				IF (bMinPosMonitoring) THEN
					lrHomingSearchMin := lrMinPos;
				ELSE
					lrHomingSearchMin := -100;
				END_IF
				IF (bMaxPosMonitoring) THEN
					lrHomingSearchMax := lrMaxPos;
				ELSE
					lrHomingSearchMax := 100;
				END_IF
				lrInitTargetSpeed := stAxisParameters.fRefVeloSearch;
				eStep := SP_RunStp1;
			SP_RunStp1 :  (* Move to homing sensor*)
				IF  NOT bHomeSensor THEN
					lrInitTargetPos := lrHomingSearchMin; (*Go in*)
					eStep := SP_RunStp2;
				ELSE
					lrInitTargetPos := lrHomingSearchMax; (*Go out*)
					eStep := SP_RunStp3;
				END_IF
				eInitCommand := AC_MoveAtAbsPos;
			SP_RunStp2 :  (*moving in, search homing*)
				IF afbMoveAbs[iUseBlock].Done THEN
					eCurrentState := AS_InPosition;
				ELSIF afbMoveAbs[iUseBlock].CommandAborted THEN
					iDebugPos := 10;
					eCurrentState := AS_InError;
				ELSIF  bHomeSensor THEN
					lrInitTargetPos := lrHomingSearchMax; (*Go out*)
					eInitCommand := AC_MoveAtAbsPos;
					eStep := SP_RunStp3;
				END_IF
			SP_RunStp3 :(* Moving out, out of sensor*)
				IF afbMoveAbs[iUseBlock].Done THEN
					eCurrentState := AS_InPosition;
				ELSIF afbMoveAbs[iUseBlock].CommandAborted THEN
					iDebugPos := 11;
					eCurrentState := AS_InError;
				ELSIF  NOT bHomeSensor THEN
					lrInitTargetPos := lrHomingSearchMin; (*Go in*)
					eInitCommand := AC_MoveAtAbsPos;
					lrInitTargetSpeed := stAxisParameters.fRefVeloSync;  (* set slow speed*)
					eStep := SP_RunStp4;
				END_IF
			SP_RunStp4 :  (*moving in slowly, search homing*)
				IF afbMoveAbs[iUseBlock].Done THEN
					eCurrentState := AS_InPosition;
				ELSIF afbMoveAbs[iUseBlock].CommandAborted THEN
					iDebugPos := 12;
					eCurrentState := AS_InError;
				ELSIF  bHomeSensor THEN
					lrHomingOffset := ABS(lrCurrentPos);
					lrInitTargetPos := lrCurrentPos; (*Go to home*)
					lrHomingPercent := (lrHomingOffset / lrUnitMotorTurn) * 100;
					eInitCommand := AC_MoveAtAbsPos;
					eStep := SP_RunStp5;
				END_IF
			SP_RunStp5 :(* Wait until position is reached *)
				IF afbMoveAbs[iUseBlock].Done THEN
					eCurrentState := AS_InPosition;
				ELSIF afbMoveAbs[iUseBlock].CommandAborted THEN
					iDebugPos := 13;
					eCurrentState := AS_InError;
				END_IF
			END_CASE
		IF NOT bAxisReady THEN
			iDebugPos := 14;
			eCurrentState := AS_InError;
		END_IF
	AS_MovingLimitNeg:
		CASE eStep OF
			SP_RunStp0 :
				IF bAxisHomed THEN
					eStep := SP_RunStp1;
				ELSE
					eStep := SP_RunStp10;
				END_IF
				lrInitTargetSpeed := stAxisParameters.fRefVeloSearch;
			SP_RunStp1 :  (* Move to Lower limit*)
				IF bMinPosMonitoring THEN
					lrInitTargetPos := lrMinPos;
					eInitCommand := AC_MoveAtAbsPos;
					eStep := SP_RunStp2;
				ELSE
					eCurrentState := AS_InPosition;
					// eCurrentState := AS_InPosition; // TODO : Code Original A enlever com. ?????
				(*ELSIF bNegLimitSwitch THEN // Modif pour test
					eCurrentState := AS_InPosition;
				ELSE
					eCommand := AC_MoveLimitNeg;*)
				END_IF
			SP_RunStp2:
				IF afbMoveAbs[iUseBlock].Done THEN
					eCurrentState := AS_OnLimitNeg;
				ELSIF afbMoveAbs[iUseBlock].CommandAborted THEN
					iDebugPos := 15;
					eCurrentState := AS_InError;
				END_IF
			SP_RunStp10 :  (* Move to LimitNeg sensor*)
				IF  bNegLimitSwitch THEN
					eStep := SP_RunStp13;
				ELSIF lrMoveOutDist = 0 THEN
					eCurrentState := AS_NotHomed;
				ELSE
					lrPosition := lrMoveOutDist+1;
					bSetPosition := TRUE;
					eStep := SP_RunStp11;
				END_IF
				eInitCommand := AC_MoveAtAbsPos;
			SP_RunStp11:
				IF fbSetPosition.Done THEN
					lrInitTargetPos := -lrMoveOutDist;
					eInitCommand := AC_MoveAtRelPos;
					eStep := SP_RunStp12;
				END_IF
			SP_RunStp12:
				IF afbMoveRel[iUseBlock].Done THEN
					eStep := SP_RunStp10;
				ELSIF afbMoveRel[iUseBlock].CommandAborted THEN
					IF  bNegLimitSwitch THEN
						eStep := SP_RunStp13;
					ELSE
						iDebugPos:= 16;
						eCurrentState := AS_InError;
					END_IF
				END_IF
			SP_RunStp13:
				IF bMinPosMonitoring THEN
					lrPosition := lrMinPos+0.5;
					bSetPosition := TRUE;
					eStep := SP_RunStp14;
				ELSE
					eCurrentState := AS_NotHomed;
				END_IF
			SP_RunStp14:
				IF fbSetPosition.Done THEN
					eCurrentState := AS_OnLimitNeg;
				END_IF
			END_CASE
		IF NOT bAxisReady THEN
			iDebugPos := 17;
			eCurrentState := AS_InError;
		END_IF
	AS_OnLimitNeg:
		CASE eCommand OF
			AC_ServoOff:
				eCurrentState := AS_PowerOff;
			AC_Home, AC_Init:
				IF bAxisHomed THEN
					eCurrentState := AS_InPosition;
				ELSE
					eCurrentState := AS_Homing;
				END_IF
		END_CASE
		IF NOT bAxisReady THEN
			iDebugPos := 18;
			eCurrentState := AS_InError;
		END_IF
	AS_Stopping:
		CASE eStep OF
			SP_RunStp0:
				iUseBlock := (iUseBlock + 1) MOD 2;
				bRemoveLimitSecurity := FALSE;
				bHome			:= FALSE;
				bMoveVel 		:= FALSE;
				bMoveAbs 		:= FALSE;
				bMoveRel 		:= FALSE;
				bMoveModulo 	:= FALSE;
				bStop 			:= TRUE;
				bHalt			:= FALSE;
				eStep := SP_RunStp1;
			SP_RunStp1:
				IF afbStop[iUseBlock].Done OR afbStop[iUseBlock].CommandAborted THEN
					iDebugPos := 19;
					eCurrentState := AS_InError;
				END_IF
		END_CASE
	AS_InError:
		CASE eStep OF
			SP_RunStp0:
				ePowerCommand := AC_None;
				bMoveToLimitNegRequest := FALSE;
				bRemoveLimitSecurity := FALSE;
				bServoOn 		:= FALSE;
				bHome			:= TRUE;
				bMoveVel 		:= FALSE;
				bMoveAbs 		:= FALSE;
				bMoveRel 		:= FALSE;
				bMoveModulo 	:= FALSE;
				bStop 			:= FALSE;
				bHalt			:= FALSE;
				bSetPosition 		:= FALSE;
				bAxisHomed		:= FALSE;
				eHomingMode	:= MC_ResetCalibration;
				eStep := SP_RunStp1;
			SP_RunStp1:
				IF fbHome.Done OR fbHome.Error THEN
					bHome := FALSE;
					eStep := SP_RunStp2;
				END_IF
			SP_RunStp2:
				IF bResetErrors THEN
					eCurrentState := AS_Resetting;
				END_IF
		END_CASE
	AS_Resetting:
		IF eCommand = AC_Init OR eCommand = AC_MoveLimitNeg THEN
			ePowerCommand := eCommand;
		END_IF
		CASE eStep OF
			SP_RunStp0:
				IF (eAxisType = AT_AX5000) THEN
					(* For this drive we must use a special drive command for reseting *)
					eStep :=SP_RunStp1;
				ELSE
					eStep :=SP_RunStp10;
				END_IF
			SP_RunStp1:
				fbResetSOE(
					Axis := sAxis,
					Execute := FALSE
				);
				fbResetSOE(
					Axis := sAxis,
					Execute := TRUE
				);
				eStep :=SP_RunStp2;
			SP_RunStp2:
				fbResetSOE(
					Axis := sAxis,
					Execute := FALSE
				);
				IF NOT fbResetSOE.Busy THEN
					IF fbResetSOE.Error THEN
						iDebugPos :=20;
						eCurrentState := AS_InError;
					ELSE
						eStep :=SP_RunStp10;
					END_IF
				END_IF
			SP_RunStp10:
				fbReset(
					Execute 		:= FALSE,
					Axis 		:= sAxis);
				fbReset(
					Execute 		:= TRUE,
					Axis 		:= sAxis);
				eStep :=SP_RunStp11;
			SP_RunStp11:
				fbReset(
					Execute 		:= FALSE,
					Axis 		:= sAxis);
				IF  NOT fbReset.Busy THEN
					IF fbReset.Error THEN
						iDebugPos :=21;
						eCurrentState := AS_InError;
					ELSE
						eCurrentState := AS_PowerOff;
					END_IF
				END_IF
		END_CASE
END_CASE

fbPower(
	Enable			:=	bServoOn,
	Enable_Positive	:=	bServoOn AND NOT bPosLimitSwitch,
	Enable_Negative	:=	bServoOn  AND NOT bNegLimitSwitch,
	Override 			:= 	100.000,
	Axis				:=	sAxis);

fbHome(
	Execute 			:= bHome,
	Position 			:= 0,
	HomingMode		:= eHomingMode,
	bCalibrationCam 	:= bHomeSensor,
	Axis 			:= sAxis);

FOR i:=0 TO 1 DO
	afbMoveAbs[i](
		Execute			:=	bMoveAbs AND iUseBlock = i,
		Position			:=	lrPosition,
		Velocity			:=	lrSpeed,
		Acceleration		:=	lrAcceleration,
		Deceleration		:=	lrDeceleration,
		Jerk 			:=	lrJerk,
		Axis				:=	sAxis);
	afbMoveModulo[i](
		Execute			:=	bMoveModulo AND iUseBlock = i,
		Position			:=	lrPosition,
		Velocity			:=	lrSpeed,
		Acceleration		:=	lrAcceleration,
		Deceleration		:=	lrDeceleration,
		Jerk 			:=	lrJerk,
		Direction    		:=	MC_Shortest_Way,
		Axis				:=	sAxis);
	afbMoveRel[i](
		Execute			:=	bMoveRel AND iUseBlock = i,
		Distance			:=	lrPosition,
		Velocity			:=	lrSpeed,
		Acceleration		:=	lrAcceleration,
		Deceleration		:=	lrDeceleration,
		Jerk 			:=	lrJerk,
		Axis				:=	sAxis);
	afbMoveVel[i](
		Execute			:=	bMoveVel AND iUseBlock = i,
		Velocity			:=	lrSpeed,
		Acceleration		:=	lrAcceleration,
		Deceleration		:=	lrDeceleration,
		Jerk 			:=	lrJerk,
		Direction			:=	eMoveDir,
		Axis				:=	sAxis);
	afbStop[i](
		Execute		:=	bStop AND iUseBlock = i,
		Deceleration	:=	lrDeceleration,
		Jerk 		:=	lrJerk,
		Axis			:=	sAxis);
	afbHalt[i](
		Execute		:=	bHalt AND iUseBlock = i,
		Deceleration	:=	lrDeceleration,
		Jerk 		:=	lrJerk,
		Axis			:=	sAxis);
END_FOR

fbSetPosition(
	Execute		:= bSetPosition,
	Position		:= lrPosition,
	Axis 		:=sAxis);
bSetPosition := FALSE;

fbReadPos(
	Enable 		:= TRUE,
	Axis 		:=sAxis);

fbReadParamTimeToGo(
	Enable 		:= TRUE,
	ReadMode 	:= READMODE_CYCLIC,
	ParameterNumber := AxisRemainingTimeToGo,
	Axis 		:=sAxis
);

(*
fbReadParamModulo(
	Enable 		:= TRUE,
	ReadMode 	:= READMODE_CYCLIC,
	ParameterNumber := AxisEncoderModuloValue,
	Axis 		:=sAxis
);

fbReadParamMinPos(
	Enable 		:= TRUE,
	ReadMode 	:= READMODE_CYCLIC,
	ParameterNumber := SWLimitNeg,
	Axis 		:=sAxis
);

fbReadParamMaxPos(
	Enable 		:= TRUE,
	ReadMode 	:= READMODE_CYCLIC,
	ParameterNumber := SWLimitPos,
	Axis 		:=sAxis
);*)
IF NOT fbReadParameters.Busy THEN
	bReadParameters := NOT bReadParameters;
END_IF

fbReadParameters(
	Execute := 	bReadParameters,
	Parameter := stReadAxisParameters,
	Axis := sAxis
);

fbReadStatus(
	Enable 		:= TRUE,
	Axis 		:=sAxis
);

IF fbReadParamTimeToGo.Valid THEN
	lrRemainingTimeToGo := fbReadParamTimeToGo.Value;
END_IF
(*
IF fbReadParamModulo.Valid THEN
	lrModuloValue := fbReadParamModulo.Value;
END_IF
IF fbReadParamMinPos.Valid THEN
	lrMinPos := fbReadParamMinPos.Value;
END_IF
IF fbReadParamMaxPos.Valid THEN
	lrMaxPos := fbReadParamMaxPos.Value;
END_IF *)
IF fbReadPos.Valid THEN
	lrCurrentPos := fbReadPos.Position;
END_IF

IF fbReadParameters.Done THEN
	stAxisParameters := stReadAxisParameters;
	lrLimitOutSpeed := stAxisParameters.fRefVeloSearch;
	lrModuloValue := stAxisParameters.fEncModuloFactor;
	lrMinPos := stAxisParameters.fEncSoftEndMin;
	lrMaxPos := stAxisParameters.fEncSoftEndMax;
	lrManualSpeed := stAxisParameters.fVeloSlowManual;
	lrFastManualSpeed := stAxisParameters.fVeloFastManual;
	lrRunningSpeed := stAxisParameters.fVeloMaximum ; (* Maximum velocity*)
	bMinPosMonitoring := WORD_TO_BOOL(stAxisParameters.bEncEnableSoftEndMinControl);
	bMaxPosMonitoring := WORD_TO_BOOL(stAxisParameters.bEncEnableSoftEndMaxControl);
	bReadParametersOnce := TRUE;
END_IF

bAxisReady := AxisIsReady(sAxis.NcToPlc.StateDWord);
IF (eAxisType = AT_AX5000) THEN
	sAxis.PlcToNc.ControlDWord := AxisSetAcceptBlockedDriveSignal(sAxis.PlcToNc.ControlDWord, bRemoveLimitSecurity);
	(* sAxis.PlcToNc.ControlDWord.8 := bRemoveLimitSecurity;  Should be remove 01.09.2016 DRE *)
END_IF

(* Error checking*)
IF AxisInErrorState(sAxis.NcToPlc.AxisState) OR fbPower.Error OR fbHome.Error OR fbSetPosition.Error OR fbReadPos.Error OR  (* fbReadParamModulo.Error OR fbReadParamMinPos.Error OR fbReadParamMaxPos.Error OR*) fbReadParameters.Error OR NOT bPowerIsOn THEN
	iDebugPos :=22;
	eCurrentState := AS_InError;
END_IF
FOR i:=0 TO 1 DO
	IF afbMoveAbs[i].Error OR afbMoveModulo[i].Error OR afbMoveRel[i].Error OR afbMoveVel[i].Error OR afbStop[i].Error OR afbHalt[i].Error THEN
		//iDebugPos :=23;
		eCurrentState := AS_InError;
	END_IF
END_FOR

(*Manual Mode Handling *)

stServoButton.Enable := bPowerIsOn AND ((eCurrentState = AS_InPosition) OR (eCurrentState = AS_NotHomed) OR (eCurrentState = AS_PowerOff) OR (eCurrentState = AS_Powering) OR (eCurrentState = AS_OnLimitNeg));
stServoButton.Activate := bServoOn;

iStep := eStep;
iState := eCurrentState;

END_FUNCTION_BLOCK

// ---- POUs/Controls/FB_CheckJack1_2.TcPOU
FUNCTION_BLOCK FB_CheckJack1_2

(*
	Description 	: Bloc fonction de test d'un vérin 1 commande, 2 capteurs
	Auteur		: DLA
	Date		: 26.03.2014
	Version		: 1.00

	Modifications :

*)

VAR_INPUT
	bJackGoOut	: BOOL;
	bJackIsIn	: BOOL;
	bJackIsOut	: BOOL;
	bResetErrors 	: BOOL;
	tTimeOut		: TIME			:= T#400ms;
END_VAR
VAR_OUTPUT
	bJackError	: BOOL;
END_VAR
VAR
	T_Error		: TON;
	RSJackErr	: RS;
	bJackErr		: BOOL;
END_VAR

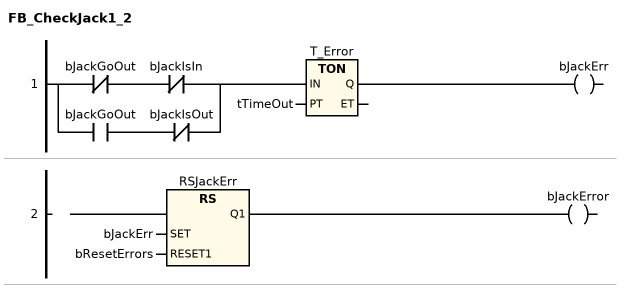
// NETWORK 1
T_Error(IN := NOT bJackGoOut AND NOT bJackIsIn OR bJackGoOut AND NOT bJackIsOut, PT := tTimeOut); // TON
bJackErr := T_Error.Q;

// NETWORK 2
RSJackErr(SET := bJackErr, RESET1 := bResetErrors); // RS
bJackError := RSJackErr.Q1;

END_FUNCTION_BLOCK

// ---- POUs/Controls/FB_VacuumAnalogCheck.TcPOU
FUNCTION_BLOCK FB_VacuumAnalogCheck

(*
	Description 	: Bloc fonction de gestion d'un module de mise sous vide avec niveau de mesure de vide analogique
	Auteur		: DRE
	Date		: 24.08.2016
	Version		: 1.00

	Modifications :

*)

VAR_INPUT
	bEnableVacuum			: BOOL	:= FALSE;			(* Demande d'activation du vacuum *)
	tBlowingTime				: TIME	:= t#200ms;			(* Temps de soufflage à la coupure du vacuum *)
	tVacErrorDelay			: TIME	:= t#400ms;			(* Temps de détection d'une erreur de vide *)
	bReset					: BOOL	:= FALSE;			(* MAZ du bloc en cas d'erreur *)
	iVacuum					: INT;						(* Capteur de vacuum *)
	tWaitVacuumOK			: TIME	:= t#0ms;				(* Temps de détection d'un vide correct *)
	lrVacuumThreshold		: LREAL	:= 9; //-0.7;				(* Seuil de dépression demandée *)
	bDisableVacuumChecking	: BOOL	:= FALSE;
END_VAR
VAR_OUTPUT
	bVacuumOn				: BOOL	:= FALSE;			(* Activation du vacuum *)
	bBlowOn					: BOOL	:= FALSE;			(* Activation du soufflage *)
	bVacuumError			: BOOL	:= FALSE;			(* La demande d'activation s'est terminée par une erreur *)
	lrVacuum				: LREAL	:= 0;					(* Dépression actuelle *)
	bVacuumOK				: BOOL;
	bVacuumCorrect			: BOOL	:= FALSE;			(* La demande d'activation a été bien traitée *)
	bVacuumStable			: BOOL	:= FALSE;			(* Le vacuum est stabilisé *)
END_VAR
VAR
	TInput					: ConverterLinearLimit;
	TVacuum				: FB_Vacuum;
END_VAR
VAR PERSISTENT
	iAnalogMinVoltage		: INT	:= 6500;				(* 1V*)
	iAnalogMaxVoltage 		: INT	:= 31600;				(*5V*)
	lrAnalogMinVacuum		: LREAL	:= 0;					(*kPa or l/min*)
	lrAnalogMaxVacuum 		: LREAL	:= 9.6;					(*kPa or l/min*)
END_VAR

TInput(
	iInput := iVacuum,
	iHardwareMin := iAnalogMinVoltage,
	iHardwareMax := iAnalogMaxVoltage,
	lrSoftwareMin := lrAnalogMinVacuum,
	lrSoftwareMax :=lrAnalogMaxVacuum
	);
lrVacuum := TInput.lrValue;
bVacuumOK := (lrVacuum <= lrVacuumThreshold) AND bEnableVacuum;			// Fonctionnement en vaccum

TVacuum(
	bEnableVacuum := bEnableVacuum,
	tBlowingTime := tBlowingTime,
	tVacErrorDelay := tVacErrorDelay,
	bReset := bReset,
	bVacuumOK := bVacuumOK,
	tWaitVacuumOK := tWaitVacuumOK,
	bDisableVacuumChecking := bDisableVacuumChecking,
	bVacuumOn => bVacuumOn,
	bBlowOn => bBlowOn,
	bVacuumError => bVacuumError,
	bVacuumCorrect => bVacuumCorrect
);

END_FUNCTION_BLOCK

// ---- POUs/utils/ConverterLinearLimit.TcPOU
FUNCTION_BLOCK ConverterLinearLimit
VAR_INPUT
	iInput			: INT;
	iHardwareMin 	: INT;
	iHardwareMax 	: INT;
	lrSoftwareMin 		: LREAL;
	lrSoftwareMax 	: LREAL;
	lrOffset			: LREAL := 0;
END_VAR
VAR_OUTPUT
	lrValue				: LREAL;
	bInputOutOfRange		: BOOL;
END_VAR
VAR
	lrMinOut 			: LREAL;
	lrMaxOut 			: LREAL;
	iHwMinIn 		: LREAL;
	iHwMaxIn		: LREAL;

END_VAR

lrValue := (

			(
				(INT_TO_LREAL(iInput) - INT_TO_LREAL(iHardwareMin))
				/
				(INT_TO_LREAL(iHardwareMax) - INT_TO_LREAL(iHardwareMin))
			)
			*
			( lrSoftwareMax - lrSoftwareMin )
		)
		+ lrSoftwareMin;
IF (lrSoftwareMin > lrSoftwareMax) THEN
	lrMinOut := lrSoftwareMax;
	lrMaxOut := lrSoftwareMin;
ELSE
	lrMinOut := lrSoftwareMin;
	lrMaxOut := lrSoftwareMax;
END_IF
IF lrValue > lrMaxOut THEN lrValue := lrMaxOut; END_IF
IF lrValue < lrMinOut THEN lrValue := lrMinOut; END_IF
lrValue := lrValue + lrOffset;

IF (iHardwareMin > iHardwareMax) THEN
	iHwMinIn := iHardwareMax;
	iHwMaxIn := iHardwareMin;
ELSE
	iHwMinIn := iHardwareMin;
	iHwMaxIn := iHardwareMax;
END_IF
bInputOutOfRange := FALSE;
IF (iInput < iHwMinIn) OR  (iInput > iHwMaxIn) THEN
	bInputOutOfRange:= TRUE;
ELSE
	bInputOutOfRange:= FALSE;
END_IF

END_FUNCTION_BLOCK

// ---- POUs/Controls/FB_Vacuum.TcPOU
FUNCTION_BLOCK FB_Vacuum

(*
	Description 	: Bloc fonction de gestion d'un module de mise sous vide
	Auteur		: DLA
	Date		: 26.03.2014
	Version		: 1.00

	Modifications :

*)

VAR_INPUT
	bEnableVacuum				: BOOL	:= FALSE;			(* Demande d'activation du vacuum *)
	tBlowingTime					: TIME	:= t#200ms;			(* Temps de soufflage à la coupure du vacuum *)
	tVacErrorDelay				: TIME	:= t#400ms;			(* Temps de détection d'une erreur de vide *)
	bReset						: BOOL	:= FALSE;			(* MAZ du bloc en cas d'erreur *)
	bVacuumOK					: BOOL;						(* Capteur de vacuum présent *)
	tWaitVacuumOK				: TIME	:= t#0ms;				(* Temps de détection d'un vide correct *)
	bDisableVacuumChecking		: BOOL	:= FALSE;
END_VAR
VAR_OUTPUT
	bVacuumOn				: BOOL	:= FALSE;			(* Activation du vacuum *)
	bBlowOn					: BOOL	:= FALSE;			(* Activation du soufflage *)
	bVacuumError			: BOOL	:= FALSE;			(* La demande d'activation s'est terminée par une erreur *)
	bVacuumCorrect			: BOOL	:= FALSE;			(* La demande d'activation a été bien traitée *)
	bVacuumStable			: BOOL	:= FALSE;			(* Le vacuum est stabilisé *)
END_VAR
VAR
	bVacuumIsOK			: BOOL	:= FALSE;			(* Information que le vacuum est OK *)
	TVacError				: TON;
	TVacOK					: TON;
	TBlow					: TON;
	TVacCut					: TON;
END_VAR

(*La commande de vacuum est directement reliée à la requête*)
bVacuumOn := bEnableVacuum;

bVacuumIsOK := bVacuumOK;

(*On fait tourner les timers de détection de vacuum et de soufflage*)
TBlow(IN:=NOT bEnableVacuum,PT:=tBlowingTime);
TVacOK(IN:=bEnableVacuum AND bVacuumOK,PT:=tWaitVacuumOK);
TVacCut(IN := NOT bEnableVacuum AND NOT bVacuumOK AND NOT bBlowOn, PT := t#100ms);
bVacuumStable := TVacOK.Q;

IF bEnableVacuum THEN
	bBlowOn := FALSE;
	(*On détecte si le vacuum ne s'établit pas assez vite*)
	TVacError(IN:=NOT (bVacuumOK OR bDisableVacuumChecking) ,PT:=tVacErrorDelay);
	IF bDisableVacuumChecking THEN
		bVacuumCorrect := TRUE;
	ELSE
		bVacuumCorrect := TVacOK.Q;
	END_IF
	IF  TVacError.Q AND NOT bVacuumOK THEN
		bVacuumError := TRUE;
	END_IF
ELSE
	(*On contrôle que le vacuum s'est bien coupé aprés le soufflage*)
	bBlowOn := NOT TBlow.Q;
	bVacuumCorrect := NOT bVacuumOK AND NOT bBlowOn;
	bVacuumCorrect := TVacCut.Q;
	TVacError(IN:=bVacuumOK AND NOT bBlowOn,PT:=tVacErrorDelay);
	IF TVacError.Q THEN
		bVacuumError := TRUE;
	END_IF
END_IF
IF bVacuumCorrect THEN
	TVacError(IN:=FALSE);
END_IF
IF bReset AND bVacuumError THEN
	TBlow(IN:= FALSE);
	TVacError(IN:=FALSE);
	bVacuumOn := FALSE;
	bBlowOn := FALSE;
	bReset := FALSE;
	bVacuumError := FALSE;
END_IF

END_FUNCTION_BLOCK

// ---- POUs/utils/ComputeVisionPos.TcPOU
FUNCTION_BLOCK ComputeVisionPos
VAR_INPUT
	THead			: TPositionXY;
	lrAngle			: LREAL;
END_VAR
VAR_OUTPUT
	TOffsetPos				: TPositionXYTheta;
END_VAR
VAR
	lrHypotenuse		: LREAL;
	lrAngle1			: LREAL;
	lrAngle2			: LREAL;
	lrAngleVision		: LREAL;
END_VAR

lrAngleVision := LMOD((lrAngle* -1) + 180 + 45,180);
lrHypotenuse := SQRT(EXPT(THead.lrX,2) + EXPT(THead.lrY,2));
IF THead.lrX = 0 THEN
	lrAngle1 := 90;
ELSE
	lrAngle1 := RAD_TO_DEG(ATAN(ABS(THead.lrY) / ABS(THead.lrX)));
END_IF
IF THead.lrX < 0 AND THead.lrY >= 0 THEN
	lrAngle1 := lrAngle1 + 90;
ELSIF THead.lrX < 0 AND THead.lrY < 0 THEN
	lrAngle1 := lrAngle1 + 180;
ELSIF THead.lrX >= 0 AND THead.lrY < 0 THEN
	lrAngle1 := lrAngle1 + 270;
END_IF
lrAngle2 := lrAngleVision - lrAngle1;
TOffsetPos.lrX := COS(DEG_TO_RAD(lrAngle2)) * -lrHypotenuse;
TOffsetPos.lrY := SIN(DEG_TO_RAD(lrAngle2)) * lrHypotenuse;
TOffsetPos.lrTheta := lrAngleVision;

END_FUNCTION_BLOCK

// ---- POUs/utils/InitNewPartData.TcPOU
FUNCTION InitNewPartData : TPartData
VAR_INPUT
END_VAR
VAR
	TPartData	: TPartData;
	i			: INT;
	j			: INT;
END_VAR

TPartData.bPartPresent := FALSE;
TPartData.bToReject := FALSE;
TPartData.bSample := FALSE;
FOR i := 0 TO 1 DO
	FOR j := 0 TO 1 DO
		TPartData.abHasPearls[i,j] := FALSE;
		TPartData.abBadPearling[i,j] := FALSE;
		TPartData.abPearlingDone[i,j] := FALSE;
		TPartData.anLastPearlIndexDone[i,j] := 0;
	END_FOR
END_FOR
TPartData.dwPlateInQRCode := 0;
TPartData.iPlateInPos := 0;
TPartData.dwPlateOutQRCode := 0;
TPartData.iPlateOutPos := 0;
TPartData.ePartSide := PS_SUS;
TPartData.dwProductionTime := 0;
TPartData.dwProductionInTime := 0;
TPartData.dwProductionOutTime := 0;
InitNewPartData := TPartData;

END_FUNCTION

// ---- POUs/utils/GetLoaderTeachedAxisFromAxis.TcPOU
FUNCTION GetLoaderTeachedAxisFromAxis : TLoaderTeachedAxis
VAR_INPUT
	eAxis	: TLoaderAxis;
END_VAR
VAR
END_VAR

CASE eAxis OF
	LA_X:
		GetLoaderTeachedAxisFromAxis := LTA_X;
	LA_Y:
		GetLoaderTeachedAxisFromAxis := LTA_Y;
	LA_Z1:
		GetLoaderTeachedAxisFromAxis := LTA_Z;
	LA_Z2:
		GetLoaderTeachedAxisFromAxis := LTA_Z;
	LA_THETA:
		GetLoaderTeachedAxisFromAxis := LTA_THETA;
END_CASE

END_FUNCTION

// ---- POUs/Handlers/TableHdl.TcPOU
FUNCTION_BLOCK TableHdl

(*
	Description 	: Function bloc to handle rotation table
	Author		: DLA
	Date		: 18.08.2014
	Version		: 1.00

	Modifications :

*)

VAR_INPUT
	bEnable						: BOOL;
	bPowerOn					: BOOL;
	bHomeTable					: BOOL;
	bHomeBrush					: BOOL;
	bLimitPosBrush				: BOOL;
	bLimitNegBrush				: BOOL;
	bResetErrors				: BOOL;
	iTableVacuumPos1Flow		: INT;
	iTableVacuumPos2Flow		: INT;
	iTableVacuumPos3Flow		: INT;
	iTableVacuumPos4Flow		: INT;
	bTableLocked				: BOOL;
	bTableNotLocked				: BOOL;
	bAspirationIsUp				: BOOL;
	bAspirationIsDown			: BOOL;
	bCheckVacuum4Rotation		: BOOL;
	eCommand					: TModuleCommands;
	bStopReq					: BOOL;
	bPauseReq					: BOOL;
	sInGiveToLoader				: TTaker;
	sInTakeFromLoader			: TGiver;
	eRunCommand				: TRunCmdTable;
	bLayeringWithTwoParts		: BOOL;
	bManInterlock				: BOOL;
	sVaccumSettings				: TVaccumSettings;
	iPartialGiveTakeTime			: INT;
	bVisionConfig					: BOOL;
	bCleanBrushIsUp				: BOOL;
	bCleanBrushIsDown				: BOOL;
END_VAR
VAR_OUTPUT
	bModuleError					: BOOL;
	bAspirationError				: BOOL;
	bIndexTableError				: BOOL;
	bPlate1VacuumError			: BOOL;
	bPlate2VacuumError			: BOOL;
	bPlate3VacuumError			: BOOL;
	bPlate4VacuumError			: BOOL;
	bTableAxisError				: BOOL;
	bBrushAxisError				: BOOL;
	bAspirationGoDown			: BOOL;
	bAspirationGoUp				: BOOL;
	bIndexTable					: BOOL;
	bAspirationBrushOn			: BOOL;
	bActivatePlate1Vacuum		: BOOL;
	bActivatePlate1Blowing		: BOOL;
	bActivatePlate2Vacuum		: BOOL;
	bActivatePlate2Blowing		: BOOL;
	bActivatePlate3Vacuum		: BOOL;
	bActivatePlate3Blowing		: BOOL;
	bActivatePlate4Vacuum		: BOOL;
	bActivatePlate4Blowing		: BOOL;
	bVacuumErrForRotation		: BOOL;
	bVacuumNotOk4Pearling		: BOOL;
	eSideOnLoader				: TTableSide;
	sOutGiveToLoader			: TGiver;
	sOutTakeFromLoader			: TTaker;
	eRunStatus					: TRunStatus;
	bManInterlockOut			: BOOL;
	aiPearlsVacuumFlow			: ARRAY[0..1] OF INT;
	bMoveCleanBrushDown			: BOOL;
	bCleanBrushError			: BOOL;
END_VAR
VAR_IN_OUT
	sCurrentState					: TModuleData;
	sRunData					: TRunDataTable;
	TManualCmd					: TManTable;
	sTableAxisRef				: AXIS_REF;
	sBrushAxisRef				: AXIS_REF;
END_VAR
VAR CONSTANT
	lrSafeTolerance 					:LREAL := 1;											(* Tolerance for safety axis *)
	lrPositionTolerance 				: LREAL := 0.1;
END_VAR
VAR PERSISTENT
	alrWorkingPos				: ARRAY [0..1] OF LREAL := [0,180];		(* Working position of table CW / CCW *)
	alrBrushParkPos				: ARRAY [0..1] OF LREAL := [0,0];
	alrBrushWorkPos				: ARRAY [0..1] OF LREAL := [90,90];
	alrBrushSpeed				: ARRAY [0..1] OF LREAL := [80,100]; 	// initial value [40,60];
	lrTableJogStep				: LREAL					:= 5;
	iNbOfCleaning				: INT					:= 1;
	lrBrushJogStep				: LREAL					:= 5;
	alrVacuumThreshold			: ARRAY[0..3] OF LREAL	:= [8,8,8,8];// [-0.65,-0.65,-0.65,-0.65];
	lrTableCleanSpeed			: LREAL					:= 30;
END_VAR
VAR
	i							: INT;
	abEnablePlateVacuum			: ARRAY[0..3] OF BOOL;
	abPlateVacuumOK			: ARRAY[0..3] OF BOOL;
	abPlateVacuumError			: ARRAY[0..3] OF BOOL;
	abForceBlowing				: ARRAY[0..3] OF BOOL;
	abDisableVacuumChecking	: ARRAY[0..3] OF BOOL;
	abActivatePlateBlowing		: ARRAY[0..3] OF BOOL;
	abActivatePlateVacuum		: ARRAY[0..3] OF BOOL;
	aiTableVacuumPosFlow	: ARRAY[0..3] OF INT;
	eMoveTableAxisCommand		: TAxisCommands	:= AC_None;
	eMoveBrushAxisCommand		: TAxisCommands	:= AC_None;
	lrTableTargetPos				: LREAL;
	lrBrushTargetPos				: LREAL;
	lrCurrentTableMoveSpeed		: LREAL;
	lrRunTableMoveSpeed		: LREAL;
	lrCurrentBrushMoveSpeed		: LREAL;
	TAspiration					: FB_CheckJack2_2;
	TIndexTable					: FB_CheckJack1_2;
	TCleanBrush				: FB_CheckJack1_2;
	aTPlateVacuum				: ARRAY[0..3] OF  FB_VacuumAnalogCheck;
	TAxisTable					: StdAxis;
	TAxisBrush					: StdAxis;
	iGiveTakePos				: INT;
	iCleaningPos					: INT;
	iCleaningCycle				: INT;
	iOffsetPosNotTakeGive		: INT;
	iTargetWorkingPos			: INT;
	TGiveTakeTimer				: TON;
	bPartialGiveTake				: BOOL;
	bTableOkToMove			: BOOL;
	TVacuumTimer				: TON;
	eLastStatus 					: TModuleStatus := MS_Stopped;
	tPartialGiveTakeTime			: TIME;
	bCleanAfterTurn				: BOOL;
	eCleaningStep				: TModuleSteps;
	bDoCleaningSeq				: BOOL;
	bDoCleaningOnMoveSeq		: BOOL;
	bStopCleaningOnMoveSeq		: BOOL;
	iStep						: INT;
END_VAR

IF (NOT sCurrentState.bStepMode) THEN
	sCurrentState.bWaitStep := FALSE;
END_IF

(* Optimize code *)
aiTableVacuumPosFlow[0] := iTableVacuumPos1Flow;
aiTableVacuumPosFlow[1] := iTableVacuumPos2Flow;
aiTableVacuumPosFlow[2] := iTableVacuumPos3Flow;
aiTableVacuumPosFlow[3] := iTableVacuumPos4Flow;
tPartialGiveTakeTime := INT_TO_TIME(iPartialGiveTakeTime);

IF eLastStatus<>sCurrentState.eStatus THEN
	IF eLastStatus=MS_Manual THEN
		(*Leave manual mode, redefine part present base on vacuum *)
		IF NOT abEnablePlateVacuum[0] THEN
			sRunData.aTPartData[0,0,TS_A].bPartPresent := FALSE;
			sRunData.aTPartData[0,1,TS_A].bPartPresent := FALSE;
		END_IF
		IF NOT abEnablePlateVacuum[1] THEN
			sRunData.aTPartData[1,0,TS_A].bPartPresent := FALSE;
			sRunData.aTPartData[1,1,TS_A].bPartPresent := FALSE;
		END_IF
		IF NOT abEnablePlateVacuum[2] THEN
			sRunData.aTPartData[0,0,TS_B].bPartPresent := FALSE;
			sRunData.aTPartData[0,1,TS_B].bPartPresent := FALSE;
		END_IF
		IF NOT abEnablePlateVacuum[3] THEN
			sRunData.aTPartData[1,0,TS_B].bPartPresent := FALSE;
			sRunData.aTPartData[1,1,TS_B].bPartPresent := FALSE;
		END_IF
	END_IF
	IF eLastStatus=MS_Running OR sCurrentState.eStatus=MS_Manual THEN
		(* Set vaccum base on part present, Vacuum can be disable if take part has failed*)
		IF NOT bVisionConfig THEN
			abEnablePlateVacuum[0] := sRunData.aTPartData[0,0,TS_A].bPartPresent OR sRunData.aTPartData[0,1,TS_A].bPartPresent;
		END_IF
		abEnablePlateVacuum[1] := sRunData.aTPartData[1,0,TS_A].bPartPresent OR sRunData.aTPartData[1,1,TS_A].bPartPresent;
		abEnablePlateVacuum[2] := sRunData.aTPartData[0,0,TS_B].bPartPresent OR sRunData.aTPartData[0,1,TS_B].bPartPresent;
		abEnablePlateVacuum[3] := sRunData.aTPartData[1,0,TS_B].bPartPresent OR sRunData.aTPartData[1,1,TS_B].bPartPresent;
	END_IF
	eLastStatus := sCurrentState.eStatus;
END_IF
IF NOT bLayeringWithTwoParts THEN
	sRunData.aTPartData[0,1,TS_A].bPartPresent := FALSE;
	sRunData.aTPartData[1,1,TS_A].bPartPresent := FALSE;
	sRunData.aTPartData[0,1,TS_B].bPartPresent := FALSE;
	sRunData.aTPartData[1,1,TS_B].bPartPresent := FALSE;
END_IF

CASE eCommand OF
	MC_NoCmd :
		CASE sCurrentState.eStatus OF
			MS_Init :
				CASE sCurrentState.eStep OF
					SP_InitStp1 :
						(* Init all synchros *)
						FOR i := 0 TO 3 DO
							abForceBlowing[i] := FALSE;
							abDisableVacuumChecking[i] := FALSE;
							(*abEnablePlateVacuum[i] := TRUE;*)
						END_FOR
						bMoveCleanBrushDown := FALSE;
						bAspirationBrushOn := FALSE;
						TVacuumTimer(IN := FALSE);
						sCurrentState.eStep := SP_InitStp2;
					SP_InitStp2 :
						TVacuumTimer(IN := TRUE, PT := t#0s);
						IF TVacuumTimer.Q THEN
							IF NOT bVisionConfig THEN
								abEnablePlateVacuum[0] := sRunData.aTPartData[0,0,TS_A].bPartPresent OR sRunData.aTPartData[0,1,TS_A].bPartPresent;
							END_IF
							abEnablePlateVacuum[1] := sRunData.aTPartData[1,0,TS_A].bPartPresent OR sRunData.aTPartData[1,1,TS_A].bPartPresent;
							abEnablePlateVacuum[2] := sRunData.aTPartData[0,0,TS_B].bPartPresent OR sRunData.aTPartData[0,1,TS_B].bPartPresent;
							abEnablePlateVacuum[3] := sRunData.aTPartData[1,0,TS_B].bPartPresent OR sRunData.aTPartData[1,1,TS_B].bPartPresent;
							IF bLayeringWithTwoParts THEN
							 	abDisableVacuumChecking[0] := sRunData.aTPartData[0,0,TS_A].bPartPresent XOR sRunData.aTPartData[0,1,TS_A].bPartPresent;
								abDisableVacuumChecking[1] := sRunData.aTPartData[1,0,TS_A].bPartPresent XOR sRunData.aTPartData[1,1,TS_A].bPartPresent;
								abDisableVacuumChecking[2] := sRunData.aTPartData[0,0,TS_B].bPartPresent XOR sRunData.aTPartData[0,1,TS_B].bPartPresent;
								abDisableVacuumChecking[3] := sRunData.aTPartData[1,0,TS_B].bPartPresent XOR sRunData.aTPartData[1,1,TS_B].bPartPresent;
							END_IF
							IF sCurrentState.bInitDone THEN
								sCurrentState.eStep := SP_InitStp50;
							ELSE
								sCurrentState.eStep := SP_InitStp3;
							END_IF
						END_IF
					SP_InitStp3 :
						(* Put the clean brush in the waiting position - Raise the aspiration - Lower index table *)
						bAspirationGoDown := FALSE;
						bIndexTable := FALSE;
						sCurrentState.eStep := SP_InitStp4;
					SP_InitStp4 :
						(* Wait until all jacks are in position *)
						IF  bAspirationIsUp AND bTableNotLocked THEN
							sCurrentState.eStep := SP_InitStp5;
						END_IF
					SP_InitStp5 :
						eMoveBrushAxisCommand := AC_Init;
						eMoveTableAxisCommand := AC_Init;
						sCurrentState.eStep := SP_InitStp6;
					SP_InitStp6 :
						IF TAxisTable.eCurrentState =  AS_InPosition AND TAxisBrush.eCurrentState =  AS_InPosition THEN
							lrTableTargetPos := alrWorkingPos[0];
							lrRunTableMoveSpeed := TAxisTable.lrRunningSpeed;
							eMoveTableAxisCommand := AC_MoveAtAbsPos;
							lrBrushTargetPos := alrBrushParkPos[0];
							(* During init always use low speed *)
							lrCurrentBrushMoveSpeed := alrBrushSpeed[0];
							eMoveBrushAxisCommand := AC_MoveAtAbsPos;
							sCurrentState.eStep := SP_InitStp7;
						END_IF
					SP_InitStp7 :
						(* Wait until init position is reached *)
						IF TAxisTable.eCurrentState =  AS_InPosition AND TAxisBrush.eCurrentState =  AS_InPosition THEN
							(* Index table *)
							bIndexTable := TRUE;
							sCurrentState.eStep := SP_InitStp8;
						END_IF
					SP_InitStp8 :
						IF bTableLocked THEN
							bAspirationGoDown := TRUE;
							sCurrentState.eStep := SP_InitStp9;
						END_IF
					SP_InitStp9 :
						IF  bAspirationIsDown THEN
							eSideOnLoader := TS_A;
							sCurrentState.eStep := SP_InitStp99;
						END_IF
					SP_InitStp50 :
						lrBrushTargetPos := alrBrushParkPos[0];
						eMoveBrushAxisCommand := AC_MoveAtAbsPos;
						sCurrentState.eStep := SP_InitStp51;
					SP_InitStp51 :
						IF TAxisBrush.eCurrentState =  AS_InPosition THEN
							sCurrentState.eStep := SP_InitStp99;
						END_IF
					SP_InitStp99 : (* Leave init *)
						sCurrentState.eStep := SP_RunStp1;
						sCurrentState.eStatus := MS_Ready;
						bDoCleaningSeq:= FALSE;
						bDoCleaningOnMoveSeq:= FALSE;
						bStopCleaningOnMoveSeq:= FALSE;
						eCleaningStep := SP_RunStp1;
						sCurrentState.bInitDone := TRUE;
				END_CASE
			MS_Running :
				IF (NOT sCurrentState.bWaitStep) THEN
					(* Cleaning sequence *)
					CASE eCleaningStep OF
						SP_RunStp1 :
							IF bUse103171OptimB5CleanOn1Move THEN
								eCleaningStep := SP_RunStp50;
							ELSE
								eCleaningStep := SP_RunStp10;
							END_IF
						SP_RunStp10 :
							IF bDoCleaningSeq THEN
								IF eSideOnLoader = TS_B THEN
									iCleaningPos := 2;
								ELSE
									iCleaningPos := 0;
								END_IF
								FOR i := 0 TO 1 DO
									IF NOT sRunData.aTPartData[i, 0, eSideOnLoader].bPartPresent AND NOT sRunData.aTPartData[i, 1, eSideOnLoader].bPartPresent THEN
										abForceBlowing[i + iCleaningPos] := TRUE;
									END_IF
								END_FOR
								bAspirationBrushOn := TRUE;
								bMoveCleanBrushDown := TRUE;
								iCleaningCycle := 0;
								eCleaningStep := SP_RunStp12;
							END_IF
						SP_RunStp11:
							IF iCleaningCycle < iNbOfCleaning THEN
								lrBrushTargetPos := alrBrushWorkPos[0];
								eMoveBrushAxisCommand := AC_MoveAtAbsPos;
								eCleaningStep := SP_RunStp12;
							ELSE
								eCleaningStep := SP_RunStp14;
							END_IF
						SP_RunStp12:
							IF (TAxisBrush.eCurrentState = AS_InPosition) THEN
								lrBrushTargetPos := alrBrushWorkPos[1];
								eMoveBrushAxisCommand := AC_MoveAtAbsPos;
								eCleaningStep := SP_RunStp13;
							END_IF
						SP_RunStp13:
							IF (TAxisBrush.eCurrentState = AS_InPosition) THEN
								iCleaningCycle := iCleaningCycle + 1;
								eCleaningStep := SP_RunStp11;
							END_IF
						SP_RunStp14:
							IF (TAxisBrush.eCurrentState = AS_InPosition) THEN
								lrBrushTargetPos := alrBrushParkPos[0];
								eMoveBrushAxisCommand := AC_MoveAtAbsPos;
								eCleaningStep := SP_RunStp15;
							END_IF
						SP_RunStp15:
							IF (TAxisBrush.eCurrentState = AS_InPosition) THEN
								eCleaningStep := SP_RunStp16;
							END_IF
						SP_RunStp16:
							FOR i := iCleaningPos TO iCleaningPos+1 DO
								abForceBlowing[i] := FALSE;
							END_FOR
							bAspirationBrushOn := FALSE;
							bMoveCleanBrushDown := FALSE;
							bDoCleaningSeq:= FALSE;
							eCleaningStep := SP_RunStp10;
						SP_RunStp50:							
							IF bDoCleaningSeq THEN
								eCleaningStep := SP_RunStp60;
							ELSIF bDoCleaningOnMoveSeq THEN
								eCleaningStep := SP_RunStp80;
							END_IF
						SP_RunStp60 :
							IF eSideOnLoader = TS_B THEN
								iCleaningPos := 1;
							ELSE
								iCleaningPos := 0;
							END_IF
							FOR i := 0 TO 1 DO
								IF NOT sRunData.aTPartData[i, 0, eSideOnLoader].bPartPresent AND NOT sRunData.aTPartData[i, 1, eSideOnLoader].bPartPresent THEN
									abForceBlowing[i + iCleaningPos] := TRUE;
								END_IF
							END_FOR
							bAspirationBrushOn := TRUE;
							bMoveCleanBrushDown := TRUE;
							eCleaningStep := SP_RunStp61;
						SP_RunStp61: 
							(* Go to other position *)
							IF TAxisBrush.lrCurrentPos < (alrBrushParkPos[0] + 1) THEN
								lrBrushTargetPos := alrBrushWorkPos[1];
							ELSE
								lrBrushTargetPos := alrBrushWorkPos[0];
							END_IF
							lrCurrentBrushMoveSpeed := alrBrushSpeed[1];
							eMoveBrushAxisCommand := AC_MoveAtAbsPos;
							eCleaningStep := SP_RunStp62;
						SP_RunStp62:
							IF (TAxisBrush.eCurrentState = AS_InPosition) THEN
								(* Move to final position *)
								lrBrushTargetPos := alrBrushWorkPos[iCleaningPos];
								eMoveBrushAxisCommand := AC_MoveAtAbsPos;
								eCleaningStep := SP_RunStp63;
							END_IF
						SP_RunStp63:
							IF (TAxisBrush.eCurrentState = AS_InPosition) THEN
								bAspirationBrushOn := FALSE;
								bMoveCleanBrushDown := FALSE;
								bDoCleaningSeq:= FALSE;
								eCleaningStep := SP_RunStp50;
							END_IF
						SP_RunStp80:
							bAspirationBrushOn := TRUE;
							bDoCleaningOnMoveSeq := FALSE;
							IF eSideOnLoader = TS_B THEN
								iCleaningPos := 0;
							ELSE
								iCleaningPos := 1;
							END_IF
							eCleaningStep := SP_RunStp81;
						SP_RunStp81:
							IF bStopCleaningOnMoveSeq THEN
								bAspirationBrushOn := FALSE;
								bStopCleaningOnMoveSeq := FALSE;
								eCleaningStep := SP_RunStp50;
							END_IF
					END_CASE
					CASE sCurrentState.eStep OF
						SP_RunStp1:
							eRunStatus := RS_WaitRequest;
							CASE eRunCommand OF
								RCT_None:
									IF bStopReq  THEN
										sCurrentState.eStatus := MS_Ready;
									ELSIF bPauseReq THEN
										sCurrentState.eStatus := MS_Paused;
									END_IF
								RCT_TakePart:
									sOutTakeFromLoader.bHasTaken := FALSE;
									sOutTakeFromLoader.bHasNotTaken := FALSE;
									sOutTakeFromLoader.bReadyToTake := TRUE;
									sCurrentState.eStep := SP_RunStp10;
								RCT_GivePart:
									sOutGiveToLoader.bHasGiven := FALSE;
									sOutGiveToLoader.bPartDataReady := FALSE;
									sCurrentState.eStep := SP_RunStp20;
								RCT_Turn:
									bCleanAfterTurn := FALSE;
									sCurrentState.eStep := SP_RunStp30;
								RCT_Clean:
									sCurrentState.eStep := SP_RunStp40;
								RCT_TurnAndClean:
									bCleanAfterTurn := TRUE;
									sCurrentState.eStep := SP_RunStp30;
							END_CASE
							IF sCurrentState.eStep<> SP_RunStp1 THEN eRunStatus := RS_ProcessRequest1; END_IF
						SP_RunStp10 :  (*Take Part*)
							IF sInTakeFromLoader.bPartDataReady THEN
								sRunData.aTPartData[ sRunData.iGiveTakeLayeringPosition, sRunData.iGiveTakeLayeringOffsetPosition, eSideOnLoader] := sInTakeFromLoader.TPartData;
								sRunData.aTPartData[sRunData.iGiveTakeLayeringPosition, sRunData.iGiveTakeLayeringOffsetPosition, eSideOnLoader].bPartPresent := FALSE;
								sCurrentState.eStep := SP_RunStp11;
							END_IF
						SP_RunStp11 :
							IF eSideOnLoader = TS_B THEN
								iGiveTakePos := sRunData.iGiveTakeLayeringPosition + 2;
							ELSE
								iGiveTakePos := sRunData.iGiveTakeLayeringPosition;
							END_IF
							iOffsetPosNotTakeGive := ((sRunData.iGiveTakeLayeringOffsetPosition + 1) MOD 2);
							abEnablePlateVacuum[iGiveTakePos] := TRUE;
							sOutTakeFromLoader.bReadyToTake := TRUE;
							IF bLayeringWithTwoParts AND NOT sRunData.aTPartData[sRunData.iGiveTakeLayeringPosition, iOffsetPosNotTakeGive, eSideOnLoader].bPartPresent THEN
								bPartialGiveTake:= TRUE;
							ELSE
								bPartialGiveTake:= FALSE;
							END_IF
							abDisableVacuumChecking[iGiveTakePos] := TRUE;
							sCurrentState.eStep := SP_RunStp12;
						SP_RunStp12 :
							(* Wait until loader has given *)
							IF sInTakeFromLoader.bHasGiven THEN
								sRunData.aTPartData[sRunData.iGiveTakeLayeringPosition, sRunData.iGiveTakeLayeringOffsetPosition, eSideOnLoader].bPartPresent := TRUE;
								abDisableVacuumChecking[iGiveTakePos] := TRUE;
								TGiveTakeTimer(IN:= FALSE);
								sCurrentState.eStep := SP_RunStp13;
							END_IF
						SP_RunStp13 :
							(* Check if the part is on Layering *)
							TGiveTakeTimer(IN:=TRUE, PT := tPartialGiveTakeTime );
							IF NOT bPartialGiveTake THEN
								IF bRejectPartWithVacuumErrorOnTable THEN
									TVacuumTimer(IN := FALSE);
									sCurrentState.eStep := SP_RunStp16;
								ELSE
									sOutTakeFromLoader.bHasTaken := TRUE;
									sCurrentState.eStep := SP_RunStp14;
								END_IF
							ELSIF TGiveTakeTimer.Q THEN
								sOutTakeFromLoader.bHasTaken := TRUE;
								sCurrentState.eStep := SP_RunStp1;
							END_IF
						SP_RunStp14 :
							IF NOT sInTakeFromLoader.bHasGiven THEN
								abDisableVacuumChecking[iGiveTakePos] := FALSE;
								sCurrentState.eStep := SP_RunStp15;
							END_IF
						SP_RunStp15 :
							IF aTPlateVacuum[iGiveTakePos].bVacuumCorrect THEN
								sCurrentState.eStep := SP_RunStp1;
							END_IF
						SP_RunStp16 :
							(* Wait until vacuum correct or vacuum error *)
							TVacuumTimer(IN := TRUE, PT := aTPlateVacuum[iGiveTakePos].tVacErrorDelay);
							IF aTPlateVacuum[iGiveTakePos].bVacuumStable THEN
								sOutTakeFromLoader.bHasTaken := TRUE;
								sCurrentState.eStep := SP_RunStp14;
							ELSIF TVacuumTimer.Q THEN
								sOutTakeFromLoader.bHasNotTaken := TRUE;
								abEnablePlateVacuum[iGiveTakePos] := FALSE;
								abDisableVacuumChecking[iGiveTakePos] := FALSE;
								sCurrentState.eStep := SP_RunStp17;
							END_IF
						SP_RunStp17 :
							IF NOT sInTakeFromLoader.bHasGiven THEN
								sRunData.aTPartData[sRunData.iGiveTakeLayeringPosition, sRunData.iGiveTakeLayeringOffsetPosition, eSideOnLoader].bPartPresent := FALSE;
								sCurrentState.eStep := SP_RunStp1;
							END_IF
						SP_RunStp20 : (*Give Part*)
							sOutGiveToLoader.TPartData := sRunData.aTPartData[sRunData.iGiveTakeLayeringPosition, sRunData.iGiveTakeLayeringOffsetPosition, eSideOnLoader];
							sOutGiveToLoader.bPartDataReady := TRUE;
							sCurrentState.eStep := SP_RunStp21;
						SP_RunStp21 :
							IF sInGiveToLoader.bReadyToTake THEN
								IF eSideOnLoader = TS_B THEN
									iGiveTakePos := sRunData.iGiveTakeLayeringPosition + 2;
								ELSE
									iGiveTakePos := sRunData.iGiveTakeLayeringPosition;
								END_IF
								abEnablePlateVacuum[iGiveTakePos] := FALSE;
								sCurrentState.eStep := SP_RunStp22;
							END_IF
						SP_RunStp22 :
							(* Check if laying vacuum is disabled *)
							IF aTPlateVacuum[iGiveTakePos].bVacuumCorrect THEN
								sOutGiveToLoader.bHasGiven := TRUE;
								sCurrentState.eStep := SP_RunStp23;
							END_IF
						SP_RunStp23 :
							(* Check if right loader has taken the plate *)
							IF sInGiveToLoader.bHasTaken THEN
								sRunData.aTPartData[sRunData.iGiveTakeLayeringPosition, sRunData.iGiveTakeLayeringOffsetPosition, eSideOnLoader].bPartPresent := FALSE;
								sCurrentState.eStep := SP_RunStp1;
							END_IF
						SP_RunStp30:
							bTableOkToMove := TRUE;
							FOR i:=0 TO 3 DO
								IF NOT aTPlateVacuum[iGiveTakePos].bVacuumCorrect THEN
									bTableOkToMove := FALSE;
								END_IF
							END_FOR
							IF bTableOkToMove THEN
								bAspirationGoDown := FALSE;
								IF bCleanAfterTurn AND bUse103171OptimB5CleanOnBothSide THEN
									bDoCleaningOnMoveSeq := TRUE;
									eCleaningStep := SP_RunStp1;
								END_IF
								sCurrentState.eStep := SP_RunStp31;
							END_IF
						SP_RunStp31 :
							IF  bAspirationIsUp THEN
								bIndexTable := FALSE;
								sCurrentState.eStep := SP_RunStp32;
							END_IF
						SP_RunStp32 :
							IF  bTableNotLocked AND NOT bDoCleaningOnMoveSeq THEN
								IF eSideOnLoader = TS_A THEN
									iTargetWorkingPos := 1;
								ELSE
									iTargetWorkingPos := 0;
								END_IF
								lrTableTargetPos := alrWorkingPos[iTargetWorkingPos];
								IF bCleanAfterTurn AND bUse103171OptimB5CleanOnBothSide THEN
									lrRunTableMoveSpeed := lrTableCleanSpeed;
								ELSE
									lrRunTableMoveSpeed := TAxisTable.lrRunningSpeed;
								END_IF
								eSideOnLoader := TS_Moving;
								eMoveTableAxisCommand := AC_MoveAtAbsPos;
								sCurrentState.eStep := SP_RunStp35;
							END_IF
						SP_RunStp35 :
							IF NOT bDoCleaningSeq THEN
								(* Wait until position is reached *)
								IF (TAxisTable.eCurrentState = AS_InPosition) THEN
									(* Index table *)
									bIndexTable := TRUE;
									(* And clean if needed *)
									IF bUse103171OptimB5CleanOnBothSide THEN
										bStopCleaningOnMoveSeq := TRUE;
									ELSIF bCleanAfterTurn THEN
										bDoCleaningSeq := TRUE;
										eCleaningStep := SP_RunStp1;
									END_IF
									sCurrentState.eStep := SP_RunStp36;
								END_IF
							END_IF
						SP_RunStp36 :
							IF bTableLocked THEN
								bAspirationGoDown := TRUE;
								sCurrentState.eStep := SP_RunStp37;
							END_IF
						SP_RunStp37 :
							IF  bAspirationIsDown THEN
								eRunStatus := RS_ProcessRequest2;
								IF NOT bDoCleaningSeq THEN
									IF iTargetWorkingPos = 0 THEN
										eSideOnLoader := TS_A;
									ELSE
										eSideOnLoader := TS_B;
									END_IF
									sCurrentState.eStep := SP_RunStp1;
								END_IF
							END_IF
						SP_RunStp40:
							IF NOT bDoCleaningSeq THEN
								bDoCleaningSeq := TRUE;
								eCleaningStep := SP_RunStp1;
								sCurrentState.eStep := SP_RunStp41;
							END_IF
						SP_RunStp41:
							IF NOT bDoCleaningSeq THEN
								sCurrentState.eStep := SP_RunStp1;
							END_IF
					END_CASE
				END_IF
			MS_Manual :
				TManualCmd.TAxisTable.Home.Enable := NOT bManInterlock AND bAspirationIsUp AND bTableNotLocked AND ((TAxisTable.eCurrentState = AS_InPosition) OR (TAxisTable.eCurrentState = AS_NotHomed));
				TManualCmd.TAxisTable.MoveBw.Enable := NOT bManInterlock AND bAspirationIsUp AND bTableNotLocked AND (TAxisTable.eCurrentState = AS_InPosition)  AND (TAxisTable.lrCurrentPos-lrTableJogStep >= TAxisTable.lrMinPos);
				TManualCmd.TAxisTable.MoveFw.Enable := NOT bManInterlock AND bAspirationIsUp AND bTableNotLocked AND (TAxisTable.eCurrentState = AS_InPosition) AND (TAxisTable.lrCurrentPos+lrTableJogStep <= TAxisTable.lrMaxPos);
				TManualCmd.TAxisTableLoading12Pos.MoveToTeach.Enable := NOT bManInterlock AND bAspirationIsUp AND bTableNotLocked AND (TAxisTable.eCurrentState = AS_InPosition) AND alrWorkingPos[0] >= TAxisTable.lrMinPos AND alrWorkingPos[0] <= TAxisTable.lrMaxPos;
				TManualCmd.TAxisTableLoading34Pos.MoveToTeach.Enable := NOT bManInterlock AND bAspirationIsUp AND bTableNotLocked AND (TAxisTable.eCurrentState = AS_InPosition) AND alrWorkingPos[1] >= TAxisTable.lrMinPos AND alrWorkingPos[1] <= TAxisTable.lrMaxPos;
				TManualCmd.TAxisTable.CurrentPos := TAxisTable.lrCurrentPos;

				TManualCmd.TAxisBrush.Home.Enable := NOT bManInterlock AND bTableLocked AND ((TAxisBrush.eCurrentState = AS_InPosition) OR (TAxisBrush.eCurrentState = AS_NotHomed));
				TManualCmd.TAxisBrush.MoveBw.Enable := NOT bManInterlock AND bTableLocked AND (TAxisBrush.eCurrentState = AS_InPosition)  AND (TAxisBrush.lrCurrentPos-lrBrushJogStep >= TAxisBrush.lrMinPos) ;
				TManualCmd.TAxisBrush.MoveFw.Enable := NOT bManInterlock AND bTableLocked AND (TAxisBrush.eCurrentState = AS_InPosition)  AND (TAxisBrush.lrCurrentPos+lrBrushJogStep <= TAxisBrush.lrMaxPos) ;
				FOR i:= 0 TO 1 DO
					TManualCmd.aTAxisBrushParkPos[i].MoveToTeach.Enable := NOT bManInterlock AND bTableLocked AND (TAxisBrush.eCurrentState = AS_InPosition)  AND alrBrushParkPos[i] >= TAxisBrush.lrMinPos AND alrBrushParkPos[i] <= TAxisBrush.lrMaxPos;
					TManualCmd.aTAxisBrushWorkPos[i].MoveToTeach.Enable := NOT bManInterlock AND bTableLocked AND (TAxisBrush.eCurrentState = AS_InPosition)  AND alrBrushWorkPos[i] >= TAxisBrush.lrMinPos AND alrBrushWorkPos[i] <= TAxisBrush.lrMaxPos;;
				END_FOR
				TManualCmd.TAxisBrush.CurrentPos := TAxisBrush.lrCurrentPos;

				TManualCmd.TAspirationDown.Enable := NOT bManInterlock AND  (((TAxisTable.eCurrentState = AS_InPosition) AND (ABS(TAxisTable.lrCurrentPos - alrWorkingPos[0])<lrPositionTolerance) OR  (ABS(TAxisTable.lrCurrentPos - alrWorkingPos[1])<lrPositionTolerance)) OR bAspirationGoDown);
				TManualCmd.TIndexTable.Enable := ((TAxisTable.eCurrentState = AS_InPosition) AND (ABS(TAxisTable.lrCurrentPos - alrWorkingPos[0])<lrPositionTolerance) OR  (ABS(TAxisTable.lrCurrentPos - alrWorkingPos[1])<lrPositionTolerance)) OR bIndexTable;

				IF bTableLocked AND eSideOnLoader = TS_Moving THEN
					IF (ABS(TAxisTable.lrCurrentPos - alrWorkingPos[0])<lrPositionTolerance) THEN
						eSideOnLoader := TS_A;
					ELSIF (ABS(TAxisTable.lrCurrentPos - alrWorkingPos[1])<lrPositionTolerance) THEN
						eSideOnLoader := TS_B;
					END_IF
				ELSIF NOT bTableLocked THEN
					eSideOnLoader := TS_Moving;
				END_IF
				FOR i:= 0 TO 3 DO
					TManualCmd.alrVaccumValue[i] := aTPlateVacuum[i].lrVacuum;
				END_FOR
				TManualCmd.TPlate1Vacuum.Enable := TAxisTable.eCurrentState <> AS_Moving AND TAxisTable.eCurrentState <> AS_Stopping AND TAxisTable.eCurrentState <> AS_Homing  AND
													TAxisBrush.eCurrentState <> AS_Moving AND TAxisBrush.eCurrentState <> AS_Stopping AND TAxisBrush.eCurrentState <> AS_Homing;
				TManualCmd.TPlate2Vacuum.Enable := TManualCmd.TPlate1Vacuum.Enable;
				TManualCmd.TPlate3Vacuum.Enable := TManualCmd.TPlate1Vacuum.Enable;
				TManualCmd.TPlate4Vacuum.Enable :=TManualCmd.TPlate1Vacuum.Enable;

				TManualCmd.TAspirationBrush.Enable := TRUE;
				TManualCmd.TCleanBrushDown.Enable := TRUE;
				bManInterlockOut := NOT (eSideOnLoader <> TS_Moving AND
								 ((TAxisBrush.lrCurrentPos <= (alrBrushParkPos[0]+lrSafeTolerance)) OR (TAxisBrush.lrCurrentPos >= (alrBrushParkPos[1]-lrSafeTolerance))) AND
								TAxisBrush.bAxisHomed AND bAspirationIsDown);


				CASE sCurrentState.eStep OF
					SP_ManualStp0 :
						// Table
						TManualCmd.TAxisTable.Home.Activate := FALSE;
						TManualCmd.TAxisTable.JogStep := lrTableJogStep;
						TManualCmd.TAxisTable.MoveBw.Activate := FALSE;
						TManualCmd.TAxisTable.MoveFw.Activate := FALSE;
						TManualCmd.TAxisTableLoading12Pos.MoveToTeach.Activate := FALSE;
						TManualCmd.TAxisTableLoading12Pos.Teach := FALSE;
						TManualCmd.TAxisTableLoading34Pos.MoveToTeach.Activate := FALSE;
						TManualCmd.TAxisTableLoading34Pos.Teach := FALSE;
						// Brush
						TManualCmd.TAxisBrush.Home.Activate := FALSE;
						TManualCmd.TAxisBrush.JogStep := lrBrushJogStep;
						TManualCmd.TAxisBrush.MoveBw.Activate := FALSE;
						TManualCmd.TAxisBrush.MoveFw.Activate := FALSE;
						FOR i:= 0 TO 1 DO
							TManualCmd.aTAxisBrushParkPos[i].MoveToTeach.Activate := FALSE;
							TManualCmd.aTAxisBrushParkPos[i].Teach := FALSE;
							TManualCmd.aTAxisBrushWorkPos[i].MoveToTeach.Activate := FALSE;
							TManualCmd.aTAxisBrushWorkPos[i].Teach := FALSE;
						END_FOR
						FOR i:= 0 TO 3 DO
							TManualCmd.alrVaccumThershold[i] := alrVacuumThreshold[i];
						END_FOR


						TManualCmd.TPlate1Vacuum.Activate := abEnablePlateVacuum[0];
						TManualCmd.TPlate2Vacuum.Activate := abEnablePlateVacuum[1];
						TManualCmd.TPlate3Vacuum.Activate := abEnablePlateVacuum[2];
						TManualCmd.TPlate4Vacuum.Activate := abEnablePlateVacuum[3];
						TManualCmd.TAspirationDown.Activate := bAspirationGoDown;
						TManualCmd.TIndexTable.Activate := bIndexTable;

						TManualCmd.TAspirationBrush.Activate := bAspirationBrushOn;
						TManualCmd.TCleanBrushDown.Activate := bMoveCleanBrushDown;
						sCurrentState.eStep := SP_ManualStp1;
					SP_ManualStp1 :
						IF bStopReq THEN
							sCurrentState.eStatus := MS_Stopped;
						ELSE
							FOR i:= 0 TO 1 DO
								TManualCmd.aTAxisBrushWorkPos[i].TeachedPos := alrBrushWorkPos[i];
								TManualCmd.aTAxisBrushParkPos[i].TeachedPos := alrBrushParkPos[i];
							END_FOR
							TManualCmd.TAxisTableLoading12Pos.TeachedPos := alrWorkingPos[0];
							TManualCmd.TAxisTableLoading34Pos.TeachedPos := alrWorkingPos[1];
							IF (lrTableJogStep <> TManualCmd.TAxisTable.JogStep) THEN
								lrTableJogStep := TManualCmd.TAxisTable.JogStep;
							END_IF
							IF TManualCmd.TAxisTableLoading12Pos.Teach THEN
								alrWorkingPos[0] := TAxisTable.lrCurrentPos;
								TManualCmd.TAxisTableLoading12Pos.Teach := FALSE;
							END_IF
							IF TManualCmd.TAxisTableLoading34Pos.Teach THEN
								alrWorkingPos[1] := TAxisTable.lrCurrentPos;
								TManualCmd.TAxisTableLoading34Pos.Teach := FALSE;
							END_IF
							IF TManualCmd.TAxisTableLoading12Pos.MoveToTeach.Activate THEN
								lrTableTargetPos := alrWorkingPos[0];
								sCurrentState.eStep := SP_ManualStp10;
							ELSIF TManualCmd.TAxisTableLoading34Pos.MoveToTeach.Activate THEN
								lrTableTargetPos := alrWorkingPos[1];
								sCurrentState.eStep := SP_ManualStp10;
							ELSIF TManualCmd.TAxisTable.MoveBw.Activate THEN
								lrTableTargetPos := TAxisTable.lrCurrentPos - lrTableJogStep;
								sCurrentState.eStep := SP_ManualStp10;
							ELSIF TManualCmd.TAxisTable.MoveFw.Activate THEN
								lrTableTargetPos := TAxisTable.lrCurrentPos + lrTableJogStep;
								sCurrentState.eStep := SP_ManualStp10;
							END_IF
							IF TManualCmd.TAxisTable.Home.Activate AND sCurrentState.eStep = SP_ManualStp1 THEN
								sCurrentState.eStep := SP_ManualStp20;
							END_IF


							IF (lrBrushJogStep <> TManualCmd.TAxisBrush.JogStep) THEN
								lrBrushJogStep := TManualCmd.TAxisBrush.JogStep;
							END_IF
							FOR i:= 0 TO 1 DO
								IF TManualCmd.aTAxisBrushParkPos[i].Teach THEN
									alrBrushParkPos[i] := TAxisBrush.lrCurrentPos;
									TManualCmd.aTAxisBrushParkPos[i].Teach := FALSE;
								END_IF
								IF TManualCmd.aTAxisBrushWorkPos[i].Teach THEN
									alrBrushWorkPos[i] := TAxisBrush.lrCurrentPos;
									TManualCmd.aTAxisBrushWorkPos[i].Teach := FALSE;
								END_IF
								IF TManualCmd.aTAxisBrushParkPos[i].MoveToTeach.Activate THEN
									lrBrushTargetPos := alrBrushParkPos[i];
									sCurrentState.eStep := SP_ManualStp15;
								ELSIF TManualCmd.aTAxisBrushWorkPos[i].MoveToTeach.Activate THEN
									lrBrushTargetPos := alrBrushWorkPos[i];
									sCurrentState.eStep := SP_ManualStp15;
								END_IF
							END_FOR
							IF TManualCmd.TAxisBrush.MoveBw.Activate THEN
								lrBrushTargetPos := TAxisBrush.lrCurrentPos - lrBrushJogStep;
								sCurrentState.eStep := SP_ManualStp15;
							ELSIF TManualCmd.TAxisBrush.MoveFw.Activate THEN
								lrBrushTargetPos := TAxisBrush.lrCurrentPos + lrBrushJogStep;
								sCurrentState.eStep := SP_ManualStp15;
							END_IF

							IF TManualCmd.TAxisBrush.Home.Activate AND sCurrentState.eStep = SP_ManualStp1 THEN
								sCurrentState.eStep := SP_ManualStp25;
							END_IF
							FOR i:= 0 TO 3 DO
								IF TManualCmd.alrVaccumThershold[i] <> alrVacuumThreshold[i] THEN
									alrVacuumThreshold[i] := TManualCmd.alrVaccumThershold[i];
								END_IF
							END_FOR

							bAspirationGoDown := TManualCmd.TAspirationDown.Activate;
							bIndexTable := TManualCmd.TIndexTable.Activate;
							abEnablePlateVacuum[0] := TManualCmd.TPlate1Vacuum.Activate;
							abEnablePlateVacuum[1] := TManualCmd.TPlate2Vacuum.Activate;
							abEnablePlateVacuum[2] := TManualCmd.TPlate3Vacuum.Activate;
							abEnablePlateVacuum[3] := TManualCmd.TPlate4Vacuum.Activate;
						END_IF
					SP_ManualStp10 : (*Move Table *)
						eMoveTableAxisCommand := AC_MoveAtAbsPos;
						sCurrentState.eStep := SP_ManualStp11;
					SP_ManualStp11:
						CASE TAxisTable.eCurrentState OF
							AS_InPosition, AS_InError:
								TManualCmd.TAxisTableLoading12Pos.MoveToTeach.Activate := FALSE;
								TManualCmd.TAxisTableLoading34Pos.MoveToTeach.Activate := FALSE;
								TManualCmd.TAxisTable.MoveFw.Activate := FALSE;
								TManualCmd.TAxisTable.MoveBw.Activate := FALSE;
								sCurrentState.eStep := SP_ManualStp1;
						END_CASE
					SP_ManualStp15: (*Move Brush *)
						eMoveBrushAxisCommand := AC_MoveAtAbsPos;
						sCurrentState.eStep := SP_ManualStp16;
					SP_ManualStp16:
						CASE TAxisBrush.eCurrentState OF
							AS_InPosition, AS_InError:
								FOR i := 0 TO 1 DO
									TManualCmd.aTAxisBrushParkPos[i].MoveToTeach.Activate := FALSE;
									TManualCmd.aTAxisBrushWorkPos[i].MoveToTeach.Activate := FALSE;
								END_FOR
								TManualCmd.TAxisBrush.MoveFw.Activate := FALSE;
								TManualCmd.TAxisBrush.MoveBw.Activate := FALSE;
								sCurrentState.eStep := SP_ManualStp1;
						END_CASE
					SP_ManualStp20 :  (* Init Table *)
						eMoveTableAxisCommand := AC_Home;
						sCurrentState.eStep := SP_ManualStp21;
					SP_ManualStp21 :
						CASE TAxisTable.eCurrentState OF
							AS_InPosition:
								lrTableTargetPos := alrWorkingPos[0];
								eMoveTableAxisCommand := AC_MoveAtAbsPos;
								sCurrentState.eStep := SP_ManualStp22;
							AS_InError:
								sCurrentState.eStep := SP_ManualStp1;
								TManualCmd.TAxisTable.Home.Activate := FALSE;
						END_CASE
					SP_ManualStp22 :
						CASE TAxisTable.eCurrentState OF
							AS_InPosition, AS_InError:
								sCurrentState.eStep := SP_ManualStp1;
								TManualCmd.TAxisTable.Home.Activate := FALSE;
						END_CASE
					SP_ManualStp25 :  (* Init Brush*)
						eMoveBrushAxisCommand := AC_Home;
						sCurrentState.eStep := SP_ManualStp26;
					SP_ManualStp26 :
						CASE TAxisBrush.eCurrentState OF
							AS_InPosition:
								lrBrushTargetPos := alrBrushParkPos[0];
								eMoveBrushAxisCommand := AC_MoveAtAbsPos;
								sCurrentState.eStep := SP_ManualStp27;
							AS_InError:
								sCurrentState.eStep := SP_ManualStp1;
								TManualCmd.TAxisBrush.Home.Activate := FALSE;
						END_CASE
					SP_ManualStp27 :(* Wait until init position is reached *)
						CASE TAxisBrush.eCurrentState OF
							AS_InPosition, AS_InError:
								sCurrentState.eStep := SP_ManualStp1;
								TManualCmd.TAxisBrush.Home.Activate := FALSE;
						END_CASE
				END_CASE
				bAspirationBrushOn := TManualCmd.TAspirationBrush.Activate;
				bMoveCleanBrushDown := TManualCmd.TCleanBrushDown.Activate;
			MS_Paused:
				IF bStopReq THEN
					sCurrentState.eStatus := MS_Ready;
				END_IF
		END_CASE
	MC_Init :
		sCurrentState.eStep := SP_InitStp1;
		sCurrentState.eStatus := MS_Init;
	MC_Run :
		sCurrentState.eStatus := MS_Running;
	MC_Manual :
		sCurrentState.bInitDone := FALSE;
		sCurrentState.eStatus := MS_Manual;
		sCurrentState.eStep := SP_ManualStp0;
	MC_Stop :
		sCurrentState.eStatus := MS_Stopped;
END_CASE


IF (NOT bPowerOn) THEN
	bAspirationGoDown := TRUE;
	bIndexTable := FALSE;
	TManualCmd.TAspirationDown.Activate := bAspirationGoDown;
	TManualCmd.TIndexTable.Activate := bIndexTable;
END_IF

IF bResetErrors THEN
	bVacuumErrForRotation := FALSE;
	sCurrentState.bInError := FALSE;
END_IF

IF (sCurrentState.eStatus <> MS_Manual) THEN
	IF (eMoveTableAxisCommand <> AC_None ) AND
		NOT bAspirationIsUp OR NOT bTableNotLocked THEN
		bTableAxisError := TRUE;
		eMoveTableAxisCommand := AC_None;
	END_IF
END_IF

(* Table Axis *)
IF (sCurrentState.eStatus = MS_Manual) THEN
	lrCurrentTableMoveSpeed := TAxisTable.lrManualSpeed;
ELSE
	lrCurrentTableMoveSpeed := lrRunTableMoveSpeed;
END_IF
TAxisTable(
	eCommand		:= eMoveTableAxisCommand,
	lrTargetPos		:= lrTableTargetPos,
	lrTargetSpeed	:= lrCurrentTableMoveSpeed,
	sAxis			:= sTableAxisRef,
	bResetErrors		:= bResetErrors,
	bHomeSensor	:= bHomeTable,
	bPowerIsOn		:= bPowerOn,
	eAxisType		:= AT_AX5000,
	stServoButton		:= TManualCmd.TAxisTable.ServoON
);
eMoveTableAxisCommand := AC_None;
bTableAxisError := (TAxisTable.eCurrentState = AS_InError);

(* Brush Axis *)
IF (sCurrentState.eStatus = MS_Manual) THEN
	lrCurrentBrushMoveSpeed := TAxisBrush.lrManualSpeed;
(*ELSE
	lrCurrentBrushMoveSpeed := TAxisBrush.lrRunningSpeed;
*)END_IF
TAxisBrush(
	eCommand		:= eMoveBrushAxisCommand,
	lrTargetPos		:= lrBrushTargetPos,
	lrTargetSpeed	:= lrCurrentBrushMoveSpeed,
	sAxis			:= sBrushAxisRef,
	bResetErrors		:= bResetErrors,
	bHomeSensor	:= bHomeBrush,
	bPowerIsOn		:= bPowerOn,
	bPosLimitSwitch	:= NOT bLimitPosBrush,
	bNegLimitSwitch	:= NOT bLimitNegBrush,
	lrMoveOutDist	:= 10,
	stServoButton		:= TManualCmd.TAxisBrush.ServoON
);
eMoveBrushAxisCommand := AC_None;
bBrushAxisError := (TAxisBrush.eCurrentState = AS_InError);

bAspirationGoUp := NOT bAspirationGoDown;
(* Check Aspiration Jack Error *)
TAspiration(
	bJackGoIn		:= bAspirationGoUp,
	bJackGoOut		:= bAspirationGoDown,
	bJackIsIn		:= bAspirationIsUp,
	bJackIsOut		:= bAspirationIsDown,
	tTimeOut			:= t#3s,
	bResetErrors		:= bResetErrors,
	bJackError		=> bAspirationError
);

(* Check Index Table Jack Error *)
TIndexTable(
	bJackGoOut		:= bIndexTable,
	bJackIsIn		:= bTableNotLocked,
	bJackIsOut		:= bTableLocked,
	tTimeOut			:= t#1s,
	bResetErrors		:= bResetErrors,
	bJackError		=> bIndexTableError
);

(* Check Aspiration Jack Error *)
TCleanBrush(
	bJackGoOut		:= bMoveCleanBrushDown,
	bJackIsIn		:= bCleanBrushIsUp,
	bJackIsOut		:= bCleanBrushIsDown,
	tTimeOut			:= t#3s,
	bResetErrors		:= bResetErrors,
	bJackError		=> bCleanBrushError
);

FOR i:= 0 TO 3 DO
	IF abForceBlowing[i] THEN
		aTPlateVacuum[i](
			bEnableVacuum	:= FALSE,
			tBlowingTime		:= ,
			tVacErrorDelay	:= INT_TO_TIME(sVaccumSettings.iErrorDelay),
			bReset			:= bResetErrors,
			iVacuum			:= 0,
		);
	ELSE
		aTPlateVacuum[i](
			bEnableVacuum		:= abEnablePlateVacuum[i],
			tVacErrorDelay		:= INT_TO_TIME(sVaccumSettings.iErrorDelay),
			tBlowingTime			:= INT_TO_TIME(sVaccumSettings.iBlowing),
			tWaitVacuumOK		:= INT_TO_TIME(sVaccumSettings.iWaitWhenVacuumOk),
			bReset				:= bResetErrors,
			iVacuum				:= aiTableVacuumPosFlow[i],
			lrVacuumThreshold	 :=  alrVacuumThreshold[i],
			bDisableVacuumChecking := abDisableVacuumChecking[i],
			bVacuumOn			=> abActivatePlateVacuum[i],
			bBlowOn				=> abActivatePlateBlowing[i],
			bVacuumError		=> abPlateVacuumError[i],
			bVacuumOK			=> abPlateVacuumOK[i]

		);
	END_IF
	IF abForceBlowing[i] THEN
		abPlateVacuumOK[i] := FALSE;
		abActivatePlateVacuum[i] := FALSE;
		abActivatePlateBlowing[i] := TRUE;
		abPlateVacuumError[i] := FALSE;
	END_IF
END_FOR

IF (bTableAxisError OR bBrushAxisError OR bAspirationError OR bCleanBrushError OR bIndexTableError OR abPlateVacuumError[0] OR abPlateVacuumError[1] OR abPlateVacuumError[2] OR abPlateVacuumError[3]) THEN
	sCurrentState.bInError := TRUE;
		IF (sCurrentState.eStatus <> MS_Manual) AND (sCurrentState.eStatus <> MS_Stopped) AND (sCurrentState.eStatus <> MS_Init) THEN
		sCurrentState.eStatus := MS_Ready;
	END_IF
END_IF

IF NOT bPowerOn OR bTableAxisError OR bBrushAxisError OR bIndexTableError THEN
	sCurrentState.bInitDone := FALSE;
	IF (sCurrentState.eStatus <> MS_Manual) THEN
		sCurrentState.eStatus := MS_Stopped;
	END_IF
END_IF

(*
IF bAspirationBrushOn AND (NOT sLoaderTakeLeftPlate.bTakerIsSafe OR NOT sLoaderTakeRightPlate.bTakerIsSafe OR NOT
		sPearlingTakeLeftPlate.bTakerIsSafe OR NOT sPearlingTakeRightPlate.bTakerIsSafe OR NOT
		sLoaderGiveLeftPlate.bGiverIsSafe OR NOT sLoaderGiveRightPlate.bGiverIsSafe) THEN
	sCurrentState.bInError := TRUE;
	bAspirationBrushOn := FALSE;
END_IF
*)

sRunData.eTableSide := eSideOnLoader;

bModuleError := sCurrentState.bInError;

sCurrentState.bInterlocked := bManInterlock AND  (sCurrentState.eStatus = MS_Manual);
sCurrentState.bRunning := (sCurrentState.eStatus = MS_Running);
IF (sCurrentState.eStatus <> MS_Running) THEN eRunStatus := RS_NotRunning; END_IF

IF (eSideOnLoader = TS_A) THEN
	aiPearlsVacuumFlow[PH_LEFT] := iTableVacuumPos3Flow;
	aiPearlsVacuumFlow[PH_RIGHT] := iTableVacuumPos4Flow;
ELSE
	aiPearlsVacuumFlow[PH_LEFT] := iTableVacuumPos1Flow;
	aiPearlsVacuumFlow[PH_RIGHT] := iTableVacuumPos2Flow;
END_IF

(* Optimize code *)
bPlate1VacuumError := abPlateVacuumError[0];
bPlate2VacuumError := abPlateVacuumError[1];
bPlate3VacuumError := abPlateVacuumError[2];
bPlate4VacuumError := abPlateVacuumError[3];
bActivatePlate1Blowing := abActivatePlateBlowing[0];
bActivatePlate2Blowing := abActivatePlateBlowing[1];
bActivatePlate3Blowing := abActivatePlateBlowing[2];
bActivatePlate4Blowing := abActivatePlateBlowing[3];
bActivatePlate1Vacuum := abActivatePlateVacuum[0];
bActivatePlate2Vacuum := abActivatePlateVacuum[1];
bActivatePlate3Vacuum := abActivatePlateVacuum[2];
bActivatePlate4Vacuum := abActivatePlateVacuum[3];

iStep := sCurrentState.eStep;

END_FUNCTION_BLOCK

// ---- POUs/Controls/FB_CheckJack2_2.TcPOU
FUNCTION_BLOCK FB_CheckJack2_2
(*
	Description 	: Bloc fonction de test d'un vérin 1 commande, 2 capteurs
	Auteur		: DLA
	Date		: 26.03.2014
	Version		: 1.00

	Modifications :

*)
VAR_INPUT
	bJackGoIn	: BOOL;
	bJackGoOut	: BOOL;
	bJackIsIn	: BOOL;
	bJackIsOut	: BOOL;
	bResetErrors 	: BOOL;
	tTimeOut		: TIME			:= T#400ms;
END_VAR
VAR_OUTPUT
	bJackError	: BOOL;
END_VAR
VAR
	T_Error		: TON;
	RSJackErr	: RS;
	bJackErr		: BOOL;
END_VAR

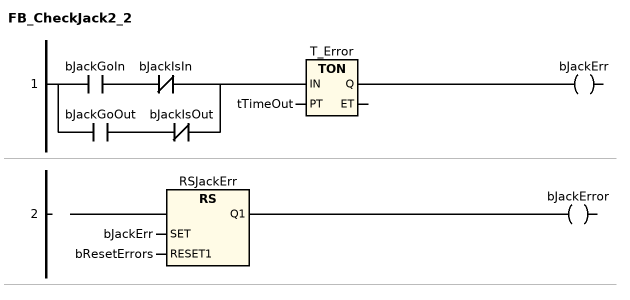
// NETWORK 1
T_Error(IN := bJackGoIn AND NOT bJackIsIn OR bJackGoOut AND NOT bJackIsOut, PT := tTimeOut); // TON
bJackErr := T_Error.Q;

// NETWORK 2
RSJackErr(SET := bJackErr, RESET1 := bResetErrors); // RS
bJackError := RSJackErr.Q1;

END_FUNCTION_BLOCK

// ---- POUs/Handlers/PearlingHdl.TcPOU
FUNCTION_BLOCK PearlingHdl

(*
	Description 	: Function bloc to handle pearling unit
	Author		: DLA
	Date		: 09.06.2014
	Version		: 1.00

	Modifications :
                                                                                                                                                                                 
*)

VAR_INPUT
	bEnable									: BOOL;										// Not used
	bPowerOn								: BOOL;										// Power activate
	eCommand								: TModuleCommands;							// Module commande
	bHomeX									: BOOL;										// Axe X Sensor home
	bLimitPosX								: BOOL;										// Axe X Sensor positif limite position
	bLimitNegX								: BOOL;										// Axe X Sensor negatif limite position
	bHomeY									: BOOL;										// Axe Y Sensor home
	bLimitPosY								: BOOL;										// Axe Y Sensor positif limite position 
	bLimitNegY								: BOOL;										// Axe Y Sensor negatif limite position 
	bHomeZ1									: BOOL;										// Axe Z1 Sensor home
	bLimitPosZ1								: BOOL;										// Axe Z1 Sensor positif limite position
	bLimitNegZ1								: BOOL;										// Axe Z1 Sensor negatif limite position
	bHomeZ2									: BOOL;										// Axe Z2 Sensor home
	bLimitPosZ2								: BOOL;										// Axe Z2 Sensor positif limite position
	bLimitNegZ2								: BOOL;										// Axe Z2 Sensor negatif limite position
	bChuck1Opened							: BOOL;										// Chuck Z1 is opened
	bChuck1Closed							: BOOL;										// Chuck Z1 is closed
	bChuck2Opened							: BOOL;										// Chuck Z2 is opened
	bChuck2Closed							: BOOL;										// Chuck Z2 is closed
	bResetErrors							: BOOL;										// Reseting the errors on the module
	bNewJob									: BOOL;										// New job loaded
	bStopReq								: BOOL;										// Request for stoping the module
	bPauseReq								: BOOL;										// Request for pausing the module
	asStickData								: ARRAY[0..1] OF TStickData;				// Description of the sticks used
	asStickDataMMI							: ARRAY[0..1] OF TStickDataMMI;				// Information for the use of the sticks from HMI
	sStickDataShared						: TStickDataShared;							// Information shared betweeen modules for the use of the sticks from HMI
	lrCompenseWeight1						: LREAL;									// Z1 weight compensation
	lrCompenseWeight2						: LREAL;									// Z2 weight compensation
	iComPort								: INT;										// 
	sInTakeFromBarrel						:TGiver;
	iContact1Distance						: INT;
	iContact2Distance						: INT;
	iLoadSensorValue						: INT;
	eSharpenRunStatus						: TRunStatus;
	eBarrelRunStatus						: TRunStatus;
	eRunCommand								: TRunCmdPearling;
	bKeepBothHeadWarm						: BOOL;
	eTableSideForLoader						: TTableSide;
	sPartData								: TPartDataMMI;
	bHead1IsUsed							: BOOL;
	bHead2IsUsed							: BOOL;
	bParallelProduction						: BOOL;
	iLeftVacuumFlow							: INT;
	iRightVacuumFlow						: INT;
	iMachineWO								: DINT;
	iMachineSN								: INT;
	yModulePosition							: BYTE;
END_VAR
VAR_OUTPUT
	bModuleError							: BOOL;
	bXAxisError								: BOOL;
	bYAxisError								: BOOL;
	bZ1AxisError							: BOOL;
	bZ2AxisError							: BOOL;
	bChuck1Error							: BOOL;
	bChuck2Error							: BOOL;
	bSpindle1Error							: BOOL;
	bSpindle2Error							: BOOL;
	bSecurityError							: BOOL;
	bSecurityErrorDetected					: BOOL;
	bMCRError								: BOOL;
	bStick1Broken							: BOOL;
	bStick2Broken							: BOOL;
	bStartPearlingMotor1					: BOOL;
	bStartPearlingMotor2					: BOOL;
	bOpenChuck1								: BOOL;
	bOpenChuck2								: BOOL;
	bActivateEject1							: BOOL;
	bActivateEject2							: BOOL;
	bActivateBlowing1						: BOOL;
	bActivateBlowing2						: BOOL;
	bAspirationPearling1On					: BOOL;
	bAspirationPearling2On					: BOOL;
	bAspirationSharpenOn					: BOOL;
	bStickContact1							: BOOL;
	bStickContact2							: BOOL;
	bCurrent1ReadError						: BOOL;
	bCurrent2ReadError						: BOOL;
	bMotor1Error							: BOOL;
	bMotor2Error							: BOOL;
	bPearlingWeight1OutOfToleranceError		: BOOL;
	bPearlingWeight2OutOfToleranceError		: BOOL;
	bStickNotTakenError						: BOOL;
	bReady2ChangeTool						: BOOL;
	iStickHead								: INT;
	sOutTakeFromBarrel						: TTaker;
	eSharpenRunCmd							: TRunCmdSharpen;
	eBarrelRunCmd							: TRunCmdBarrel;
	eRunStatus								: TRunStatus;
	bManInterlockOut						: BOOL;
	adwMotorRunningHours					: ARRAY[0..1] OF DWORD;
	adwSpindleRunningHours					: ARRAY[0..1] OF DWORD;
	bLeftSpindleUsedWarning					: BOOL;
	bRightSpindleUsedWarning				: BOOL;
	bLeftMotorUsedWarning					: BOOL;
	bRightMotorUsedWarning					: BOOL;
	bLeftSpindleLimitWarning				: BOOL;
	bRightSpindleLimitWarning				: BOOL;
	bLeftSpindleHeatWarning					: BOOL;
	bRightSpindleHeatWarning				: BOOL;
END_VAR
VAR_IN_OUT
	sCurrentState							: TModuleData;
	TManualCmd								: TManPearling;
	sRecData								: ComBuffer;
	sTransData								: ComBuffer;
	asPearlData								: ARRAY[0..1] OF TMMIPearlData;
	sXAxisRef								: AXIS_REF;
	sYAxisRef								: AXIS_REF;
	sZ1AxisRef								: AXIS_REF;
	sZ2AxisRef								: AXIS_REF;
	sRunData								: TRunDataPearling;
	asProbingLog							: ARRAY[0..1] OF  TProbingLog;
END_VAR
VAR PERSISTENT
	alrHighDynParams						: ARRAY[0..3] OF TDynAxisParam;
	alrLowDynParams							: ARRAY[0..3] OF TDynAxisParam;
	alrSafePos								: ARRAY[0..3] OF LREAL;
	alrRobotPos								: ARRAY[0..3,0..PTP_END] OF LREAL;					(* XYZ1Z2 for Ref/Inner/Outer/Drop/... *)
	alrJogStep								: ARRAY[0..3] OF LREAL;								(* Jog step for X,Y,Z1,Z2 *)
	lrSharpeningDelta						: LREAL								:= 10;
	lrSharpenPosOffset						: LREAL								:= 2;
	alrChuckRetractOffset					: ARRAY[0..1] OF LREAL				:= [1,1];		// TODO: HFO, modifier valeur, original [2, 2]
	lrStickTakeSpeed						: LREAL								:= 10;
	bBypassMCR								: BOOL;
(*	iMaxNbOfFwBwSharpen						: INT	:= 1;*)
	TBreakStickDetectTime					: TIME	:= t#30ms;
	aiContactThresholdArea					: ARRAY[0..1, 0..PA_END] OF INT;
	aiSpindleManualSpeed					: ARRAY[0..1] OF INT;
	alrSensorRate							: ARRAY[0..1] OF LREAL								(* in Unit / mm *);
	lrSensorZSpeed							: LREAL								:= 0.1;
	alrLoadSensorOffset						: ARRAY[0..1] OF LREAL;
	lrLoadSensorRate						: LREAL								:= 6.36121;			(* in Unit / g *)
	iLoadSensorTare							: INT								:= 3175;		(* in Unit / g *)
	alrRatiog2mm							: ARRAY[0..1] OF LREAL				:= [2(0.001)];
	lrStickErrorDeltaPos					: LREAL								:= 0.5;
(*	lrSpindelOffsetX						: LREAL								:= 50.0;*)
	iMCROffsetCurrent						: ARRAY[0..1] OF INT				:= [0,0];
	iMCRCurrentRatio						: ARRAY[0..1] OF INT				:= [1,1];
	aiMotorStartedTimeout					: ARRAY[0..1] OF INT 				:= [2000,2000]; (* in ms *)
	aiMotorStoppedTimeout					: ARRAY[0..1] OF INT 				:= [2000,2000]; (* in ms *)
	bForceProbing							: BOOL;
	lrStickOutAfterChange					: LREAL 							:= 12; 			(* mm *)
	lrProbingThreshold						: LREAL								:= 0.05; 		(* mm *)
	alrSharpenTeachZOffset					: LREAL								:= 0.4;
	dwMaxSpindleRunningHours				: DWORD								:= 900;			(*Hours : Max time running spindle before changing it *)
	dwMaxMotorRunningHours					: DWORD								:= 2000;		(*Hours : Max time running motor before changing it *)
	iMCRMinThCurrent						: INT								:= 200;
	iMCRMaxThCurrent 						: INT								:= 800;
	iMCRWarnThCurrent 						: INT								:= 600;
	adwPearlsCounter 						: ARRAY[0..1] OF DWORD				:= [2(0)];
	lrCenterSharpningOffset 				: LREAL 							:= 1.5;
	lrSecurityPreRefPosZ					: LREAL 							:= 1.5;
END_VAR
VAR CONSTANT
	lrLoadSensorStep						: LREAL								:= 0.02;
	lrWeightCalibrationStartOffsetZ			: LREAL 							:= 0.1;
	lrSafeTolerance 						: LREAL 							:= 1;			(* Tolerance for safety Z axis down *)
	lrMaxXYMoveAllowed						: LREAL 							:= 30;			(* Max move authorized when Z axis is down *)
	lrManMaxXYMoveAllowed					: LREAL 							:= 2.1;			(* Max move in manual mode authorized when Z axis is down *)
	lrSecurityRadius						: LREAL								:= 18;
	bInvertX								: BOOL 								:= FALSE;
	bInvertY								: BOOL 								:= FALSE;
	bInvertZ								: BOOL 								:= TRUE;
	lrLayeringCenterOffsetXTable			: LREAL 							:= 65;
	lrLayeringCenterOffsetYTable			: LREAL 							:= 18;
	iHeatOnSpeed							: INT								:= 1000;
END_VAR
VAR
	alrMaxRobotSpeed						: ARRAY[0..3] OF LREAL;
	alrManualRobotSpeed						: ARRAY[0..3] OF LREAL;
	i										: INT;
	j										: INT;
	iAxis									: INT;
	iCurrentManAxis							: INT;
	eRobotXYStatus							: TAxisState;
	aeMoveRobotCommand						: ARRAY[0..3] OF TAxisCommands		:= [4(AC_None)];
	aTRobotAxis								: ARRAY[0..3] OF StdAxis;
	alrCurrentSpeed							: ARRAY[0..3] OF LREAL;
	alrTargetPos							: ARRAY[0..3] OF LREAL;
(*	abForceNewPosZ							: ARRAY[0..1] OF BOOL;*)
	nPearlIndex								: UINT;
	aTPearlingTimer							: ARRAY[0..1] OF TON;
	TCheckTimer								: TON;
	alrPreRefPosZ							: ARRAY[0..1] OF LREAL;
(*	bRemoveXLimitSecurity					: BOOL;
	bRemoveYLimitSecurity					: BOOL;*)
	bManualZIsSafe							: BOOL;
	abChangeStick							: ARRAY[0..1] OF BOOL				:= [TRUE,TRUE];
	abSharpenStick							: ARRAY[0..1] OF BOOL				:= [TRUE,TRUE];
	abDoProbing								: ARRAY[0..1] OF BOOL;
	abRetryProbing							: ARRAY[0..1] OF BOOL;
	abProbingDone							: ARRAY[0..1] OF BOOL;
	aiProbingCount							: ARRAY[0..1] OF INT;
	alrProbingStartPos						: ARRAY[0..1] OF LREAL;
	eStickStep								: TModuleSteps;
	aeProbingStep							: ARRAY[0..1] OF TModuleSteps;
	TCheckTime								: TIME								:= T#5S;
	TMCRDrv									: MCRDrv;
	aTCheckChuck							: ARRAY[0..1] OF FB_CheckJack1_2;
	alrCorrectionMCR						: ARRAY[0..1] OF LREAL;
	eMCRCommand								: TMCRCommands;
	bMCRReady								: BOOL;
(*	abLastStickContact						: ARRAY[0..1] OF BOOL;*)
	aiNbOfPearlsDone						: ARRAY[0..1] OF INT;
	iCurrentArea							: INT;
	aArea									: ARRAY[0..C_MAX_NB_OF_PEARLS] OF TPearlsArea;
	alrPearlingEnergy						: ARRAY[0..1] OF LREAL;
	aTDispersion							: ARRAY[0..1] OF Dispersion;
	alrRemainingStickLength					: ARRAY[0..1] OF LREAL;
	aTMotorCounter							: ARRAY[0..1] OF RunningCounter;
	aTSpindleCounter						: ARRAY[0..1] OF RunningCounter;
	TWaitChuckOpen							: TON;
	abZRefTaken								: ARRAY[0..3,0..1,0..1] OF BOOL; 					(*Layring , Offset Layring, Head *)
	alrSecurityPosition						: ARRAY[0..3,0..1,0..1] OF LREAL;					(*Layring , Offset Layring, Head *)
	alrContactPosition						: ARRAY[0..3,0..1,0..1] OF LREAL;					(*Layring , Offset Layring, Head *)
	alrContactStickPosition					: ARRAY[0..3,0..1,0..1] OF LREAL;					(*Layring , Offset Layring, Head *)
	alrProbingRef							: ARRAY[0..3,0..1,0..1] OF LREAL; 					(*Layring , Offset Layring, Head *)
	alrHeadSecurityPosition					: ARRAY[0..1] OF LREAL;
	alrHeadContactPosition					: ARRAY[0..1] OF LREAL;
	alrHeadContactStickPosition				: ARRAY[0..1] OF LREAL;
	alrHeadProbingRef						: ARRAY[0..1] OF LREAL;
	alrSharpenProbing						: ARRAY[0..1] OF LREAL;
	alrDeltaSharpenProbing					: ARRAY[0..1] OF LREAL;
	alrStickCorrection						: ARRAY[0..1] OF LREAL;
	alrDeltaStickCorrection					: ARRAY[0..1] OF LREAL;
	alrFirstPearlCorrection					: ARRAY[0..1] OF LREAL;
	abTakeZRef								: ARRAY[0..1] OF BOOL;
	bClearZRef								: BOOL;
	abNeedSharpening						: ARRAY[0..1] OF BOOL;
	abNeedChangeStick						: ARRAY[0..1] OF BOOL;
	bFirstStart								: BOOL								:= TRUE;
	bFirstInit								: BOOL								:= TRUE;
	abBadPearling							: ARRAY[0..1] OF BOOL;
	alrDynParams							: ARRAY[0..3] OF TDynAxisParam;
	yMCRChannel								: BYTE;
	abPearlStarted							: ARRAY[0..1] OF BOOL;
	abPearlDone								: ARRAY[0..1] OF BOOL;
	abPearlPosReached						:  ARRAY[0..1] OF BOOL;
	lrRadius								: LREAL;
	alrLastProbingPos						: ARRAY[0..1] OF LREAL;
	aTWaitMotorStarted						: ARRAY[0..1] OF TON;
	aTWaitMotorStopped						: ARRAY[0..1] OF TON;
	iNbOfFwBwSharpen						: INT;
	iNbOfFwBwSharpenBeforeMove				: INT;
	abNewStick								: ARRAY[0..1] OF BOOL				:= [FALSE,FALSE];
	iDebugPos								: INT;
	iDebugSide								: INT;
	aTDetectStickBroken						: ARRAY[0..1] OF TON;
(*	bZIsSafe								: BOOL;*)
	alrProbingPos							: ARRAY[0..1] OF LREAL;
	alrCheckProbingPos						: ARRAY[0..1] OF LREAL;
	alrProbingLimit							: ARRAY[0..1] OF LREAL;
(*	iNbOfPearlsRemainingOnThisArea			: INT;*)
	abCheckingStick							: ARRAY[0..1] OF BOOL;
	TWaitCurrentMotorBeltOk					: TON;
	TWaitCurrentMotorWarmOk					: TON;
	aTStickContactValidated					: ARRAY[0..1] OF TON;
	TStickContactValidTime					: TIME								:= T#250MS; // valeur original ==> t#500ms; Temps de stabilisation du capteur de de distance en contacte
	TStickStabilisationTime					: TIME								:= T#400MS;	// Temps pour stabiliser le capteur de distance sans contact
	aIMinPos								: ARRAY[0..1] OF INT;
	alrDeltaZPearl							: ARRAY[0..1] OF LREAL;
	alrDeltaWeightPearl						: ARRAY[0..1] OF LREAL;
	iTableIndex								: INT;
	lrBasePos								: LREAL;
(*	TWaitEjectorTimer						: TON;*)
	abWeightTableValid						: ARRAY[0..1] OF BOOL;
	alrWeightTable							: ARRAY[0..1,0..C_WEIGHT_TABLE_MAX] OF LREAL;
	iSide									: INT;
	abStartPearlingMotor					: ARRAY[0..1] OF BOOL;
	aiContactDistance						: ARRAY[0..1] OF INT;
	abUseSpindle							: ARRAY[0..1] OF BOOL;
	abChuckOpened							: ARRAY[0..1] OF BOOL;
	abChuckClosed							: ARRAY[0..1] OF BOOL;
	abOpenChuck								: ARRAY[0..1] OF BOOL;
	abActivateEject							: ARRAY[0..1] OF BOOL;
	abSpindleError							: ARRAY[0..1] OF BOOL;
	abAspirationPearling					: ARRAY[0..1] OF BOOL;
	abStickContact							: ARRAY[0..1] OF BOOL;
	abActivateBlowing						: ARRAY[0..1] OF BOOL;
	abCurrentReadError						: ARRAY[0..1] OF BOOL;
	abMotorError							: ARRAY[0..1] OF BOOL;
	abSpindleCurrentOk						: ARRAY[0..1] OF BOOL;
	abStickBroken							: ARRAY[0..1] OF BOOL;
	abStickBrokenDetected					: ARRAY[0..1] OF BOOL;
	abPearlNeeded							: ARRAY[0..1] OF BOOL;
	abHeadIsUsed							: ARRAY[0..1] OF BOOL;
	abPearlingWeightOutOfToleranceError		: ARRAY[0..1] OF BOOL;
	abPearlingWeightOutOfToleranceDetected	: ARRAY[0..1] OF BOOL;
	abFirstPearl							: ARRAY[0..1] OF BOOL;
	aiCountPearlError						: ARRAY[0..1] OF INT;
	alrBasePearlingEnergy					: ARRAY[0..1] OF LREAL;
	alrCompenseWeight						: ARRAY[0..1] OF LREAL;
	aiPearlingLayringPos					: ARRAY[0..1] OF INT;
	aiPearlingLayringOffsetPos				: ARRAY[0..1] OF INT;
	anPearlIndexDone						: ARRAY[0..1] OF UINT;
	aiSideInfo								: ARRAY[0..1] OF INT;
	TLayeringCenter							:  TPositionXY;
	TPearlPosition							:  TPositionXY;
	iFirstHeadUsed							: INT;
	iRejectPos								: INT;
	iChangeStickPos							: INT;
	nPearl									: UINT;
	aiPearlingTeachedPos					: ARRAY[0..1] OF INT;
	alrPearlingOffset						: ARRAY[0..4] OF LREAL;
	alrPearlingInvert						: ARRAY[0..4] OF LREAL;
	alrHeadPushed_mm						: ARRAY[0..1] OF LREAL;
(*	psPartData								: ARRAY[0..1] OF POINTER TO TPartData;*)
	bChangeToolSide							: BOOL;
(*	bChangeTool								: BOOL;*)
	bEndPearling							: BOOL;
	lrWeight								: LREAL;
	lrMaxMCRCorrection						: LREAL;
	bCalibrationInProgress					: BOOL;
	aeProbingArea							: ARRAY[0..1] OF TProbingArea;
	TDebug									: TPearlingDebug;
	aePearlingArea							: ARRAY[0..1] OF TProbingArea;
	TWaitHeadStab							: TON;
	atStickValidateTime						: ARRAY[0..1] OF LREAL;
	aiVacuumFlow							: ARRAY[0..1] OF INT;
	ayChannelStatus							: ARRAY[0..1] OF BYTE;
	abCurrentLimitWarning					: ARRAY[0..1] OF BOOL;
	aTWaitSpindleHeatOn						: ARRAY[0..1] OF TON;
	aTDetectSpindleCooled					: ARRAY[0..1] OF TON;
	abNeedSpindleHeatOn						: ARRAY[0..1] OF BOOL;
	ai_ProbingStep							: ARRAY [0..1] OF INT;
	i_StickStep								: INT;
	iDebugPosBrokenStick					: INT;
END_VAR


(*_AppInfo.BootDataLoaded;			// HFO, to know if boot data was loaded
_AppInfo.OldBootData;
_AppInfo.PersistentStatus;*)

(* Optimize code *)
abStartPearlingMotor[PH_Left] := bStartPearlingMotor1;
abStartPearlingMotor[PH_Right] := bStartPearlingMotor2;
aiContactDistance[PH_Left] := iContact1Distance;
aiContactDistance[PH_Right] := iContact2Distance;
abChuckOpened[PH_Left] := bChuck1Opened;
abChuckOpened[PH_Right] := bChuck2Opened;
abChuckClosed[PH_Left] := bChuck1Closed;
abChuckClosed[PH_Right] := bChuck2Closed;
alrCompenseWeight[PH_Left] := lrCompenseWeight1;
alrCompenseWeight[PH_Right] := lrCompenseWeight2;
abHeadIsUsed[PH_Left] := bHead1IsUsed;
abHeadIsUsed[PH_Right] := bHead2IsUsed;
aiVacuumFlow[PH_LEFT] := iLeftVacuumFlow;
aiVacuumFlow[PH_RIGHT] := iRightVacuumFlow;

eSharpenRunCmd := RCS_None;
eBarrelRunCmd := RCB_None;

IF bInvertX THEN
	alrPearlingInvert[PA_X] := -1;
ELSE
	alrPearlingInvert[PA_X] := 1;
END_IF
IF bInvertY THEN
	alrPearlingInvert[PA_Y] := -1;
ELSE
	alrPearlingInvert[PA_Y] := 1;
END_IF
IF bInvertZ THEN
	alrPearlingInvert[PA_Z1] := -1;
	alrPearlingInvert[PA_Z2] := -1;
ELSE
	alrPearlingInvert[PA_Z1] := 1;
	alrPearlingInvert[PA_Z2] := 1;
END_IF

FOR iAxis := 0 TO 3 DO
	alrMaxRobotSpeed[iAxis] := aTRobotAxis[iAxis].lrRunningSpeed;
	alrManualRobotSpeed[iAxis] := aTRobotAxis[iAxis].lrManualSpeed;
END_FOR

IF (NOT sCurrentState.bStepMode) THEN
	sCurrentState.bWaitStep := FALSE;
END_IF

IF bFirstStart THEN
	FOR iSide := 0 TO 1 DO
		abWeightTableValid[iSide] := FALSE;
		aTDetectSpindleCooled[iSide](IN := FALSE);
		aTWaitSpindleHeatOn[iSide](IN := FALSE);
		abNeedSpindleHeatOn[iSide] := TRUE;
	END_FOR
	bFirstStart := FALSE;
END_IF

IF bNewJob THEN
	FOR iSide := 0 TO 1 DO
		abSharpenStick[iSide] := TRUE;
		aiNbOfPearlsDone[iSide] := 1;
	END_FOR
	bClearZRef := TRUE;
END_IF

FOR iSide:=0 TO 1 DO
	abStickContact[iSide] := aiContactDistance[iSide] > (aiContactThresholdArea[iSide , aeProbingArea[iSide]] + 0.05 * alrSensorRate[iSide]);
	aTWaitMotorStarted[iSide](IN := abStartPearlingMotor[iSide],PT := INT_TO_TIME(aiMotorStartedTimeout[iSide]));
	aTWaitMotorStopped[iSide](IN := NOT abStartPearlingMotor[iSide],PT := INT_TO_TIME(aiMotorStoppedTimeout[iSide]));
	aTMotorCounter[iSide](bStart := abStartPearlingMotor[iSide], bReset := FALSE);
	aTSpindleCounter[iSide](bStart := abStartPearlingMotor[iSide], bReset := FALSE);
	IF NOT abDoProbing[iSide] THEN
		abProbingDone[iSide] := FALSE;
	END_IF
	(* For debug purpose *)
	IF alrSensorRate[iSide] <> 0 THEN
		alrHeadPushed_mm[iSide] := INT_TO_REAL(LREAL_TO_INT(((aiContactDistance[iSide]-aiContactThresholdArea[iSide , aeProbingArea[iSide]])/alrSensorRate[iSide])*100))/100.0;
	ELSE
		alrHeadPushed_mm[iSide] := 0;
	END_IF
	alrBasePearlingEnergy[iSide] := sRunData.sPearlingData.iWeight +  alrCompenseWeight[iSide];
	IF bParallelProduction THEN
		aiSideInfo[iSide] := 0;
	ELSE
		aiSideInfo[iSide] := iSide;
	END_IF
END_FOR

(* For debug purpose *)
IF lrLoadSensorRate<>0 THEN
	lrWeight := (INT_TO_LREAL(iLoadSensorValue) - INT_TO_LREAL(iLoadSensorTare)) / lrLoadSensorRate;
ELSE
	lrWeight := 0;
END_IF

CASE eCommand OF
	MC_NoCmd :
		CASE sCurrentState.eStatus OF
			MS_Init :
				CASE sCurrentState.eStep OF
(*----------------- Init ------------------*)
					SP_InitStp1 :
						FOR iSide := 0 TO 1 DO
							abAspirationPearling[iSide] := FALSE;
							abActivateEject[iSide] := FALSE;
							(* Move Z Up *)
							aeMoveRobotCommand[PA_Z1+iSide] := AC_MoveLimitNeg;
						END_FOR
						bAspirationSharpenOn := FALSE;
						alrCurrentSpeed := alrMaxRobotSpeed;
						sCurrentState.eStep := SP_InitStp2;
					SP_InitStp2 :
						IF aTRobotAxis[PA_Z1].eCurrentState = AS_OnLimitNeg  AND
						     aTRobotAxis[PA_Z2].eCurrentState = AS_OnLimitNeg THEN
							(* Init X / Y*)
							aeMoveRobotCommand[PA_X] := AC_Init;
							aeMoveRobotCommand[PA_Y] := AC_Init;
							sCurrentState.eStep := SP_InitStp3;
						END_IF
					SP_InitStp3 :
						IF 	(aTRobotAxis[PA_X].eCurrentState = AS_InPosition) AND
							(aTRobotAxis[PA_Y].eCurrentState = AS_InPosition) THEN
							(* Move X/ Y to Safe *)
							alrTargetPos[PA_X] := alrSafePos[PA_X];
							alrTargetPos[PA_Y] := alrSafePos[LA_Y];
							aeMoveRobotCommand[PA_X] := AC_MoveAtAbsPos;
							aeMoveRobotCommand[PA_Y] := AC_MoveAtAbsPos;
							sCurrentState.eStep := SP_InitStp4;
						END_IF
					SP_InitStp4 :
						IF aTRobotAxis[PA_X].eCurrentState = AS_InPosition AND
						     aTRobotAxis[PA_Y].eCurrentState = AS_InPosition THEN
								(* Init Z *)
								aeMoveRobotCommand[PA_Z1] := AC_Init;
								aeMoveRobotCommand[PA_Z2] := AC_Init;
								sCurrentState.eStep := SP_InitStp5;
						END_IF
					SP_InitStp5 :
						IF aTRobotAxis[PA_Z1].eCurrentState=AS_InPosition AND
							aTRobotAxis[PA_Z2].eCurrentState=AS_InPosition THEN
							(* Move Z to Safe *)
							alrTargetPos[PA_Z1] := alrSafePos[PA_Z1];
							alrTargetPos[PA_Z2] := alrSafePos[LA_Z2];
							aeMoveRobotCommand[PA_Z1] := AC_MoveAtAbsPos;
							aeMoveRobotCommand[PA_Z2] := AC_MoveAtAbsPos;
							sCurrentState.eStep := SP_InitStp6;
						END_IF
					SP_InitStp6 :
						IF  aTRobotAxis[PA_Z1].eCurrentState = AS_InPosition AND
						     aTRobotAxis[PA_Z2].eCurrentState = AS_InPosition THEN
							IF bBypassMCR THEN
								sCurrentState.eStep := SP_InitStp99;
							ELSIF bMCRReady THEN
								yMCRChannel := 1;
								sCurrentState.eStep := SP_InitStp10;
							END_IF
						END_IF
					SP_InitStp10 :
						(* Configure MCR *)
						eMCRCommand := MCRC_ConfigMeasure;
						sCurrentState.eStep := SP_InitStp11;
					SP_InitStp11 :
						IF bMCRReady THEN
							IF yMCRChannel = 1 THEN
								yMCRChannel := 2;
								sCurrentState.eStep := SP_InitStp10;
							ELSE
								yMCRChannel := 1;
								sCurrentState.eStep := SP_InitStp12;
							END_IF
						END_IF
					SP_InitStp12 :
						eMCRCommand := MCRC_SetRatio;
						TMCRDrv.lrRatio := asStickDataMMI[yMCRChannel - 1].lrMCRRatio;
						sCurrentState.eStep := SP_InitStp13;
					SP_InitStp13 :
						IF bMCRReady THEN
							IF yMCRChannel = 1 THEN
								yMCRChannel := 2;
								sCurrentState.eStep := SP_InitStp12;
							ELSE
								yMCRChannel := 1;
								sCurrentState.eStep := SP_InitStp14;
							END_IF
						END_IF
					SP_InitStp14 :
						(* Do spindle heat on if needed *)
						TMCRDrv.iSpeedSetpoint := iHeatOnSpeed;;
						eMCRCommand := MCRC_SetSpeed;
						sCurrentState.eStep := SP_InitStp15;
					SP_InitStp15 :
						IF bMCRReady THEN
							IF yMCRChannel = 1 THEN
								yMCRChannel := 2;
								sCurrentState.eStep := SP_InitStp14;
							ELSE
								yMCRChannel := 1;
								sCurrentState.eStep := SP_InitStp16;
							END_IF
						END_IF
					SP_InitStp16 :
						abStartPearlingMotor[PH_Left] := abNeedSpindleHeatOn[PH_Left];
						abStartPearlingMotor[PH_Right] := abNeedSpindleHeatOn[PH_Right];
						sCurrentState.eStep := SP_InitStp17;
					SP_InitStp17 :
						IF (NOT (abNeedSpindleHeatOn[PH_Left] AND abStartPearlingMotor[PH_Left]) AND 
								NOT (abNeedSpindleHeatOn[PH_Right] AND abStartPearlingMotor[PH_Right])) THEN
							sCurrentState.eStep := SP_InitStp25;
						END_IF
					SP_InitStp25 :
						eMCRCommand := MCRC_SetSpeed;
						TMCRDrv.iSpeedSetpoint := sStickDataShared.sStickDataMMIShared.iMCRSharpenSpeed;
						sCurrentState.eStep := SP_InitStp26;
					SP_InitStp26 :
						IF bMCRReady THEN
							IF yMCRChannel = 1 THEN
								yMCRChannel := 2;
								sCurrentState.eStep := SP_InitStp25;
							ELSE
								yMCRChannel := 1;
								sCurrentState.eStep := SP_InitStp27;
							END_IF
						END_IF
					SP_InitStp27:
						(* Set Parameter*)
						IF NOT bFirstInit THEN
							eMCRCommand := MCRC_SetParam;
							TMCRDrv.iOffsetCurrent := iMCROffsetCurrent[yMCRChannel - 1];
							TMCRDrv.iCurrentRatio := iMCRCurrentRatio[yMCRChannel - 1];
						END_IF
						sCurrentState.eStep := SP_InitStp28;
					SP_InitStp28:
						IF bMCRReady THEN
							IF yMCRChannel = 1 THEN
								yMCRChannel := 2;
								sCurrentState.eStep := SP_InitStp27;
							ELSE
								yMCRChannel := 1;
								sCurrentState.eStep := SP_InitStp29;
							END_IF
						END_IF
					SP_InitStp29:
						(* Set threshold*)
						eMCRCommand := MCRC_DefineCurrentThr;
						TMCRDrv.iMinThCurrent := iMCRMinThCurrent;
						TMCRDrv.iMaxThCurrent := iMCRMaxThCurrent;
						TMCRDrv.iWarnThCurrent := iMCRWarnThCurrent;
						sCurrentState.eStep := SP_InitStp30;
					SP_InitStp30:
						IF bMCRReady THEN
							IF yMCRChannel = 1 THEN
								yMCRChannel := 2;
								sCurrentState.eStep := SP_InitStp29;
							ELSE
								yMCRChannel := 1;
								sCurrentState.eStep := SP_InitStp31;
							END_IF
						END_IF
					SP_InitStp31:
						IF NOT bFirstInit THEN
							(* Set MachineID*)
							eMCRCommand := MCRC_DefineMachineID;
							TMCRDrv.iMachineWO := iMachineWO;
							TMCRDrv.iMachineSN := iMachineSN;
							TMCRDrv.yMachineSide := asc('a') + yModulePosition;
						END_IF
						sCurrentState.eStep := SP_InitStp32;
					SP_InitStp32:
						IF bMCRReady THEN
							IF yMCRChannel = 1 THEN
								yMCRChannel := 2;
								sCurrentState.eStep := SP_InitStp31;
							ELSE
								yMCRChannel := 1;
								sCurrentState.eStep := SP_InitStp99;
							END_IF
						END_IF
					SP_InitStp50: (*Init if already init done, always move Z to safe *)
						(* Go to safe position *)
						alrCurrentSpeed := alrMaxRobotSpeed;
						alrTargetPos[PA_Z1] := alrSafePos[PA_Z1];
						alrTargetPos[PA_Z2] := alrSafePos[PA_Z2];
						aeMoveRobotCommand[PA_Z1] := AC_MoveAtAbsPos;
						aeMoveRobotCommand[PA_Z2] := AC_MoveAtAbsPos;
						sCurrentState.eStep := SP_InitStp51;
					SP_InitStp51 :
						IF 	(aTRobotAxis[PA_Z1].eCurrentState = AS_InPosition) AND
							(aTRobotAxis[PA_Z2].eCurrentState = AS_InPosition) THEN
							sCurrentState.eStep := SP_InitStp99;
						END_IF
					SP_InitStp99 :
						bFirstInit := FALSE;
						FOR iSide := 0 TO 1 DO
							abDoProbing[iSide] := FALSE;
							abUseSpindle[iSide] := FALSE;
							abRetryProbing[iSide] := FALSE;
							aiProbingCount[iSide] := 0;
						END_FOR
						sCurrentState.eStatus := MS_Ready;
						sCurrentState.bInitDone := TRUE;
						sCurrentState.eStep := SP_RunStp1;
						eStickStep := SP_RunStp1;
						aeProbingStep[PH_Left] := SP_RunStp1;
						aeProbingStep[PH_Right] := SP_RunStp1;

